--- mnuSetTargetPts.pgx ---
program mnuSetTargetPts()
  local bool LbBackup
  local num LnNewValue
  local string LsNameKeeper
  local num nKey
begin
  //header begin
  // PROGRAM mnuSetTargetPts()
  //
  // runs the menu to query user for all info needed to teach Target Frames/Points
  // with user input of Azimuth, Elevation, & Radius
  // output to X, Y, Z, RX, RY, RZ
  //
  // incoming parms:  none
  // outgoing parms:  none
  // called from:  pgm mnuTeachMenu()
  //
  //  initial release KN
  //header end
  //
  // start continuous loop, end by menu command or teach pendant command
  // on user command, jump to other subroutines for action
  //
  // init booleans for menu control in pgm displayMessage2()
  LbBackup=false
  bWorldFrameView=true
  //
  do
    //nIdxSetTargetPt=261
    call displayMessage2(nIdxSetTargetPt,nKey)
    // verify selection
    switch nKey
      // ESC key aborts, return with no save to pgm mnuTeachMenu()
      case 255
        return
      break
      // menu = Set Target Points
      // F1 to change Interaction Point number 0 or 1
      case 271
        nIPNumber=nIPNumber+1
        if nIPNumber==2
          nIPNumber=0
        endIf
      break
      // menu = Set Target Points
      // F2 to increment point number 0-19 in selected frame 0-1
      case 272
        if nIPNumber==0
          nIP1Number=nIP1Number+1
          if nIP1Number==20
            nIP1Number=0
          endIf
        else
          nIP2Number=nIP2Number+1
          if nIP2Number==20
            nIP2Number=0
          endIf
        endIf
      break
      // menu = Set Target Points, F3 to change the POINT NAME string
      // save currently selected name string to temporary variable
      // get new name string, test for >18 characters
      case 273
        gotoxy(19,3)
        put("                  ")
        gotoxy(19,3)
        if nIPNumber==0
          LsNameKeeper=sIP1TargName[nIP1Number]
          get(sIP1TargName[nIP1Number])
          if (len(sIP1TargName[nIP1Number])>18)
            popUpMsg("Name:  18 characters max...press OK")
            sIP1TargName[nIP1Number]=LsNameKeeper
          endIf
        else
          LsNameKeeper=sIP2TargName[nIP2Number]
          get(sIP2TargName[nIP2Number])
          if (len(sIP2TargName[nIP2Number])>18)
            popUpMsg("Name:  18 characters max...press OK")
            sIP2TargName[nIP2Number]=LsNameKeeper
          endIf
        endIf
        libSave()
      break
      //  menu = Set Target Points
      //  F4 ot change POINT AZIMUTH
      case 274
        // test input value for valid range
        LnNewValue=0
        gotoxy(26,4)
        get(LnNewValue)
        if LnNewValue>180 or LnNewValue<-180
          popUpMsg("ERROR:  Azimuth must be between 180 & -180 degrees...Press OK")
        else
          if nIPNumber==0
            nIP1Azimuth[nIP1Number]=LnNewValue
            //update Target Point to new AZ data
            call makePntAZELRA(nIPNumber,nIP1Number)
          else
            nIP2Azimuth[nIP2Number]=LnNewValue
            // update Target Point to new AZ data
            call makePntAZELRA(nIPNumber,nIP2Number)
          endIf
        endIf
        libSave()
      break
      // menu = Set Target Points
      // F5 to change POINT ELEVATION
      case 275
        // test input value for valid range
        LnNewValue=0
        gotoxy(26,5)
        get(LnNewValue)
        if LnNewValue>90 or LnNewValue<-90
          popUpMsg("ERROR:  Elevation must be between 90 & -90 degrees...Press OK")
        else
          if nIPNumber==0
            nIP1Elevation[nIP1Number]=LnNewValue
            // update Target Point to new EL data
            call makePntAZELRA(nIPNumber,nIP1Number)
          else
            nIP2Elevation[nIP2Number]=LnNewValue
            // update Target Point to new EL data
            call makePntAZELRA(nIPNumber,nIP2Number)
          endIf
        endIf
        libSave()
      break
      //  menu = Set Target Point (frame) Target Point
      //  F6 to change POINT RADIUS
      case 276
        //test input value for valid range
        LnNewValue=0
        gotoxy(26,6)
        get(LnNewValue)
        if LnNewValue<0
          popUpMsg("ERROR:  Negative Radius Disallowed...Press OK")
        else
          if nIPNumber==0
            nIP1Radius[nIP1Number]=LnNewValue
            // update Target Point to new RA data
            call makePntAZELRA(nIPNumber,nIP1Number)
          else
            nIP2Radius[nIP2Number]=LnNewValue
            // update Target Point to new RA data
            call makePntAZELRA(nIPNumber,nIP2Number)
          endIf
        endIf
        libSave()
      break
      // menu = Set Target Points, F7 to change displayed trsf values relative to the selected IP or World CoordSys
      // this boolean is acted upon in pgm displayMessage2()
      case 277
        if bWorldFrameView==true
          bWorldFrameView=false
        else
          bWorldFrameView=true
        endIf
      break
      //  menu = Set Target Points, F8 to save library on exit & return to pgm mnuTeachMenu()
      case 278
        libSave()
        LbBackup=true
      break
      // Any other key press
      default
        cls()
        popUpMsg("BAD SELECTION...press OK")
      break
    endSwitch
  until (false or (LbBackup==true))
  //
  // done
end

--- mnuTeachCube.pgx ---
program mnuTeachCube()
  local bool LbBackup
  local bool LbCubeAllDone
  local bool LbErrCreateCube
  local bool LbSetXYZdone
  local num LnXKeeper
  local num LnYKeeper
  local num LnZKeeper
  local point LpHere
  local string LsMoveMsg
  local num nKey
begin
  //header begin
  // PROGRAM mnuTeachCube()
  //
  // runs the menu to query user for all info needed to teach a Cubic Stay Clear Zone
  //
  // incoming parms:  none
  // outgoing parms:  none
  // called from:  pgm mnuTeachStyClr()
  //
  //  initial release KN
  //header end
  //
  // start continuous loop, end by menu command or teach pendant command
  // on user command, jump to other subroutines for action
  //
  // init booleans for menu control in pgm displayMessage1()
  LbBackup=false
  bCubeStep1=true
  bSetCylinderRZ=false
  bCylinderStep1=false
  bSetSphereRad=false
  bSphereStep1=false
  bSetCubeXYZ=false
  LbCubeAllDone=false
  // retrieve initial Cube data & store to temp variables for manipulation & display
  pOriginCube=MON:pOriginCube[nNumberCube]
  nDistXCube=MON:nDistXCube[nNumberCube]
  nDistYCube=MON:nDistYCube[nNumberCube]
  nDistZCube=MON:nDistZCube[nNumberCube]
  do
    //=========step 1==================step 1===============step 1================
    // Teach Cube, Step 1:  Tell user select and/or modify cube definitions
    do
      //nIdxTeachCube=201
      call displayMessage1(nIdxTeachCube,nKey)
      // verify selection
      switch nKey
        // ESC key aborts & returns immediately
        case 255
          return
        break
        // Teach Cube, F1 to ACCEPT definition & return to pgm mnuTeachStyClr()
        case 271
          LbCubeAllDone=true
          bSetCubeXYZ=false
          MON:nNumberCube=nNumberCube
          call MON:createCube(pOriginCube,nDistXCube,nDistYCube,nDistZCube,LbErrCreateCube)
          if LbErrCreateCube==true
            popUpMsg("Create Cube Failed...NO RECOVERY...Press OK")
            LbCubeAllDone=false
          endIf
          // saved at bottom
        break
        // menu = Teach Cube, F3 Button, change cube number via increment only
        // max = 10 as initially implemented in monitorAreaEn() library
        // max value change requires manual coordination, not automatic
        case 273
          nNumberCube=nNumberCube+1
          if nNumberCube==10
            nNumberCube=0
          endIf
          pOriginCube=MON:pOriginCube[nNumberCube]
          nDistXCube=MON:nDistXCube[nNumberCube]
          nDistYCube=MON:nDistYCube[nNumberCube]
          nDistZCube=MON:nDistZCube[nNumberCube]
        break
        // menu = Teach Cube, F4 Button, Tell user to Teach Origin Point
        case 274
          LsMoveMsg="Move SensorTool to Cube #"+toString("2.0",nNumberCube)+" Origin Point...OK to Teach"
          popUpMsg(LsMoveMsg)
          pOriginCube=here(tSensorTool,world)
        break
        //  menu = Teach Cube, F5 Button, Define DX, DY, DZ values
        case 275
          bSetCubeXYZ=true
          bCubeStep1=false
        break
        // menu = Teach Cube, F7 to reset this cube definition to {0, 0, 0}
        // this disables checking on this cube
        case 277
          MON:pOriginCube[nNumberCube].trsf={0,0,0,0,0,0}
          MON:nDistXCube[nNumberCube]=0
          MON:nDistYCube[nNumberCube]=0
          MON:nDistZCube[nNumberCube]=0
          pOriginCube.trsf={0,0,0,0,0,0}
          nDistXCube=0
          nDistYCube=0
          nDistZCube=0
          MON:nNumberCube=nNumberCube
          MON:bCreateCube[nNumberCube]=false
          MON:libSave()
          popUpMsg("CubeZone "+toString(".0",nNumberCube)+" CLEARED...Press OK")
        break
        // menu = Teach Cube, F8 Button, ABORT to Teach Stay Clear Zone Menu
        case 278
          bCubeStep1=false
          return
        break
        // Any other key press
        default
          cls()
          popUpMsg("BAD SELECTION...press OK")
        break
      endSwitch
    until (false or (bSetCubeXYZ==true) or (LbCubeAllDone==true))
    //
    //====step 2==============step 2===================step 2===============
    // menu = Teach Cube Step 2:  set the DX DY DZ values if required
    // Cube DX, DY, DZ values set here are temp to this pgm
    // only saved permanently in MON library on formal SAVE (F1) in above Step1
    if bSetCubeXYZ==true
      LbSetXYZdone=false
      do
        //nIdxSetCubeXYZ=211
        call displayMessage1(nIdxSetCubeXYZ,nKey)
        // verify selection
        switch nKey
          // ESC key aborts & returns immediately
          case 255
            return
          break
          // user accepts input from step 2 and auto backup to previous menu for acceptance
          case 271
            LbSetXYZdone=true
            bCubeStep1=true
          break
          case 274
            // user enters a new value for Cube DX
            gotoxy(25,6)
            LnXKeeper=nDistXCube
            get(nDistXCube)
            if (nDistXCube<0)
              popUpMsg("Negative values for Cube DX not allowed...Press OK")
              nDistXCube=LnXKeeper
            endIf
          break
          // user enters a new value for Cube DY
          case 275
            gotoxy(25,7)
            LnYKeeper=nDistYCube
            get(nDistYCube)
            if (nDistYCube<0)
              popUpMsg("Negative values for Cube DY not allowed...Press OK")
              nDistYCube=LnYKeeper
            endIf
          break
          // user enters a new value for Cube DZ
          case 276
            gotoxy(25,8)
            LnZKeeper=nDistZCube
            get(nDistZCube)
            if nDistZCube<0
              popUpMsg("Negative values for Cube DZ not allowed...Press OK")
              nDistZCube=LnZKeeper
            endIf
          break
          // ABORT to Teach Stay Clear Zone Menu menu and return to pgm mnuTeachStyClr()
          case 278
            bCubeStep1=false
            return
          break
          default
            popUpMsg("BAD SELECTION...Press OK")
          break
        endSwitch
      until (false or (LbSetXYZdone==true))
    endIf
    bSetCubeXYZ=false
    LbSetXYZdone=false
    //
  until (false or (LbCubeAllDone==true))
  bCubeStep1=false
  //
  // Teach Cube completed, save data on Exit
  libSave()
  MON:libSave()
  //
  //done
end

--- mnuTeachCyl.pgx ---
program mnuTeachCyl()
  local bool LbBackup
  local bool LbCylAllDone
  local bool LbErrCreateCyl
  local bool LbSetCylRZdone
  local num LnRKeeper
  local num LnZKeeper
  local point LpHere
  local string LsMoveMsg
  local num nKey
begin
  //header begin
  // PROGRAM mnuTeachCyl()
  //
  // runs the menu to query user for all info needed to teach a Cylinder Stay Clear Zone
  //
  // incoming parms:  none
  // outgoing parms:  none
  // called from:  pgm mnuTeachStyClr()
  //
  //  initial release KN
  //header end
  //
  // start continuous loop, end by menu command or teach pendant command
  // on user command, jump to other subroutines for action
  //
  // init booleans for menu control here & in displayMessage1()
  LbBackup=false
  bSetCubeXYZ=false
  bCubeStep1=false
  bSphereStep1=false
  bSetSphereRad=false
  bSetCylinderRZ=false
  bCylinderStep1=true
  LbCylAllDone=false
  // retrieve initial Cylinder data and store to temp variables for manipulation & display
  pOriginCylinder=MON:pOriginCylinder[nNumberCylinder]
  nRadiusCylinder=MON:nRadiusCylinder[nNumberCylinder]
  nDistZCylinder=MON:nDistZCylinder[nNumberCylinder]
  do
    //=========step 1==================step 1===============step 1================
    // menu = Teach Cylinder, Step 1:  Main Cylinder Info Display
    do
      //nIdxTeachCyl=221
      call displayMessage1(nIdxTeachCyl,nKey)
      // verify selection
      switch nKey
        // ESC key aborts & returns immediately
        case 255
          return
        break
        // Teach Cylinder, F1 to ACCEPT definition & return to pgm mnuTeachStyClr()
        case 271
          LbCylAllDone=true
          bSetCylinderRZ=false
          MON:nNumberCylinder=nNumberCylinder
          call MON:createCylinder(pOriginCylinder,nRadiusCylinder,nDistZCylinder,LbErrCreateCyl)
          if LbErrCreateCyl==true
            popUpMsg("Create Cylinder Failed...NO RECOVERY...Press OK")
            LbCylAllDone=false
          endIf
          // saved at bottom
        break
        // menu = Teach Cylinder, F3 Button, change cylinder number via increment only
        // max = 10 as initially implemented in monitorAreaEn() library
        // max value change requires manual coordination, not automatic
        case 273
          nNumberCylinder=nNumberCylinder+1
          if nNumberCylinder==10
            nNumberCylinder=0
          endIf
          pOriginCylinder=MON:pOriginCylinder[nNumberCylinder]
          nRadiusCylinder=MON:nRadiusCylinder[nNumberCylinder]
          nDistZCylinder=MON:nDistZCylinder[nNumberCylinder]
        break
        // menu = Teach Cylinder, F4 Button, Tell user to Teach Origin Point
        case 274
          LsMoveMsg="Move robot to Cylinder #"+toString("2.0",nNumberCylinder)+" Origin Point...OK to Teach"
          popUpMsg(LsMoveMsg)
          pOriginCylinder=here(tSensorTool,world)
        break
        //  menu = Teach Cylinder, F5 Button, goto Step2 to Define Radius & DZ values
        case 275
          bSetCylinderRZ=true
          bCylinderStep1=false
        break
        // menu = Teach Cylinder, F7 to reset this cylinder definition to {0,0,0}
        // this disables checking of this cylinder volume
        case 277
          MON:pOriginCylinder[nNumberCylinder].trsf={0,0,0,0,0,0}
          MON:nRadiusCylinder[nNumberCylinder]=0
          MON:nDistZCylinder[nNumberCylinder]=0
          pOriginCylinder.trsf={0,0,0,0,0,0}
          nRadiusCylinder=0
          nDistZCylinder=0
          MON:nNumberCylinder=nNumberCylinder
          MON:bCreateCylinder[nNumberCube]=false
          MON:libSave()
          popUpMsg("CylinderZone "+toString(".0",nNumberCylinder)+" CLEARED...Press OK")
        break
        // menu = Teach Cylinder, F8 Button, ABORT & Backup
        case 278
          bCylinderStep1=false
          return
        break
        // Any other key press
        default
          cls()
          popUpMsg("BAD SELECTION...press OK")
        break
      endSwitch
    until (false or (bSetCylinderRZ==true) or (LbCylAllDone==true))
    //
    //====step 2==============step 2===================step 2===============
    // menu = Teach Cylinder Step 2:  set the Radius & DZ values if required
    // Cylinder DZ & Radius values here are temp to this pgm
    // only saved permanently in MON library on formal SAVE (F1) in above Step1
    if bSetCylinderRZ==true
      LbSetCylRZdone=false
      do
        //nIdxSetCylRZ=231
        call displayMessage1(nIdxSetCylRZ,nKey)
        // verify selection
        switch nKey
          // ESC key aborts & returns immediately
          case 255
            return
          break
          // user accepts Cylinder Radius & Z-Distance input from step 2 and...
          // auto backup to previous menu for acceptance
          case 271
            LbSetCylRZdone=true
            bCylinderStep1=true
          break
          case 274
            // user enters a new value for Cylinder Radius
            gotoxy(30,6)
            LnRKeeper=nRadiusCylinder
            get(nRadiusCylinder)
            if (nRadiusCylinder<0)
              popUpMsg("Negative values disallowed...Press OK")
              nRadiusCylinder=LnRKeeper
            endIf
          break
          // user enters a new value for Cylinder DZ
          case 275
            gotoxy(25,7)
            LnZKeeper=nDistZCylinder
            get(nDistZCylinder)
            if nDistZCylinder<0
              popUpMsg("Negative values disallowed...Press OK")
              nDistZCylinder=LnZKeeper
            endIf
          break
          // menu Teach Cylinder, F7 to clear this cylinder definition
          // this disables checking of this cylinder volume
          case 277
            MON:pOriginCylinder[nNumberCylinder].trsf={0,0,0,0,0,0}
            MON:nRadiusCylinder[nNumberCylinder]=0
            MON:nDistZCylinder[nNumberCylinder]=0
            pOriginCylinder.trsf={0,0,0,0,0,0}
            nRadiusCylinder=0
            nDistZCylinder=0
            MON:nNumberCylinder=nNumberCylinder
            MON:libSave()
          break
          // ABORT & backup to previous menu
          case 278
            bCylinderStep1=false
            return
          break
          // any other key press
          default
            cls()
            popUpMsg("BAD SELECTION...Press OK")
          break
        endSwitch
      until (false or (LbSetCylRZdone==true))
    endIf
    bSetCylinderRZ=false
    LbSetCylRZdone=false
    //
  until (false or (LbCylAllDone==true))
  bCylinderStep1=false
  //
  // Teach Cylinder completed, save data on exit
  //
  libSave()
  MON:libSave()
  //
  // done
end

--- mnuTeachFrame.pgx ---
program mnuTeachFrame()
  local bool LbTeachFrm1of5
  local bool LbTeachFrm2of5
  local bool LbTeachFrm3of5
  local bool LbTeachFrm4of5
  local bool LbTeachFrm5of5
  local point LpFrameOrigin
  local point LpFrameXAxis
  local point LpFrameYAxis
  local num nKey
begin
  //header begin
  // PROGRAM mnuTeachFrame()
  //
  // runs the Wizard to assist user:  Teach the Target Frame of the two targets
  //
  // incoming parms:  none
  // outgoing parms:  none
  // called from:  pgm mnuTeachIP()
  //
  //  initial release KN
  //  Release 2 KN
  //    this pgm now called from pgm mnuTeachIP()
  //
  //header end
  //
  // start continuous loop, go through each of 5 wizard steps
  //
  // init step-by-step continuance booleans
  LbTeachFrm1of5=false
  LbTeachFrm2of5=false
  LbTeachFrm3of5=false
  LbTeachFrm4of5=false
  LbTeachFrm5of5=false
  //
  // menu = Teach Interaction Point Frame, Step 1 of 5 Steps:  select the frame to be taught
  do
    // nIdxFrm1of5=131
    call displayMessage(nIdxFrm1of5,nKey)
    // verify selection
    switch nKey
      // ESC aborts & returns immediately
      case 255
        return
      break
      // menu = Teach Interaction Point Frame 1of5, F1 to continue to Step 2 of 4
      case 271
        LbTeachFrm1of5=true
      break
      // menu = Teach Interaction Point Frame 1of5, F3 Button, user changes Target Number
      case 273
        if nIPNumber==1
          nIPNumber=-1
        else
          nIPNumber=nIPNumber+1
        endIf
      break
      // menu = Teach Interaction Point Frame 1of5, F8 Button, ABORT & backup to Teach Menu
      case 278
        return
      break
      // Any other key press
      default
        popUpMsg("BAD SELECTION...press OK")
      break
    endSwitch
  until (false or (LbTeachFrm1of5==true))
  //
  // menu = Teach Interaction Point Frame, Step 2 of 5 Steps:  verify Ref Pointer tool is attached
  do
    // nIdxFrm2of5=141
    call displayMessage(nIdxFrm2of5,nKey)
    // verify selection
    switch nKey
      // ESC key aborts & returns immediately
      case 255
        return
      break
      // menu = Teach Interaction Point Frame 2of5, F1 to continue to Step 3 of 5
      case 271
        LbTeachFrm2of5=true
      break
      // menu = Teach Interaction Point Frame 2of5, F8 Button, ABORT & backup to Teach Menu
      case 278
        return
      break
      // Any other key press
      default
        popUpMsg("BAD SELECTION...press OK")
      break
    endSwitch
  until (false or (LbTeachFrm2of5==true))
  //
  // menu = Teach Interaction Point Frame, Step 3 of 5 Steps:  move to Frame Origin
  do
    // nIdxFrm3of5=151
    call displayMessage(nIdxFrm3of5,nKey)
    // verify selection
    switch nKey
      // ESC key aborts & returns immediately
      case 255
        return
      break
      // menu = Teach Interaction Point Frame 3of5, F1 Button, teach frame origin point
      case 271
        LpFrameOrigin=here(tRefPointer,world)
        LbTeachFrm3of5=true
      break
      // menu = Teach Interaction Point Frame 3of5, F8 Button, ABORT & backup to Teach Menu
      case 278
        return
      break
      // Any other key press
      default
        popUpMsg("BAD SELECTION...press OK")
      break
    endSwitch
  until (false or (LbTeachFrm3of5==true))
  //
  // menu = Teach Interaction Point Frame, Step 4 of 5 Steps:  teach Frame X-Axis location
  do
    // nIdxFrm4of5=161
    call displayMessage(nIdxFrm4of5,nKey)
    // verify selection
    switch nKey
      // ESC key aborts & returns immediately
      case 255
        return
      break
      // menu = Teach Interaction Point Frame 4of5, F1 Button, teach Frame X-Axis point
      case 271
        LpFrameXAxis=here(tRefPointer,world)
        LbTeachFrm4of5=true
      break
      // menu = Teach Interaction Point Frame 4of5, F8 Button, ABORT & backup to Teach Menu
      case 278
        return
      break
      // Any other key press
      default
        popUpMsg("BAD SELECTION...press OK")
      break
    endSwitch
  until (false or (LbTeachFrm4of5==true))
  //
  // menu = Teach Interaction Point Frame, Step 5 of 5 Steps:  Teach Frame y-Axis direction point
  do
    // nIdxFrm5of5=171
    call displayMessage(nIdxFrm5of5,nKey)
    // verify selection
    switch nKey
      // ESC key aborts & returns immediately
      case 255
        return
      break
      // menu = Teach Interaction Point Frame 5of5, F1 Button, User Accepts Frame definition
      case 271
        LpFrameYAxis=here(tRefPointer,world)
        if nIPNumber==-1
          setFrame(LpFrameOrigin,LpFrameXAxis,LpFrameYAxis,fIPoriginal)
        elseIf nIPNumber==0
          setFrame(LpFrameOrigin,LpFrameXAxis,LpFrameYAxis,fIP1)
        elseIf nIPNumber==1
          setFrame(LpFrameOrigin,LpFrameXAxis,LpFrameYAxis,fIP2)
        endIf
        LbTeachFrm5of5=true
      break
      // menu = Teach Interaction Point Frame 5of5, F8 Button, ABORT & backup to Teach Menu
      case 278
        return
      break
      // Any other key press
      default
        popUpMsg("BAD SELECTION...press OK")
      break
    endSwitch
  until (false or (LbTeachFrm5of5==true))
  //
  // teach Interaction Point Frame completed, save data on exit
  libSave()
  //
  // done
end

--- mnuTeachIP.pgx ---
public program mnuTeachIP()
  local bool LbBackup
  local num nKey
begin
  //header begin
  // PROGRAM mnuTeachP()
  //
  // runs the menu to Teach the Interaction Point by two methods:
  //    (1) Direct Entry of Interaction Point {X, Y, Z, RX, RY, RZ} values
  //    (2) Use a Wizard to walk through the steps to physically teach the IP with a reference pointer tool
  //
  // incoming parms:  none
  // outgoing parms:  none
  // called from:  pgm mnuTeachMenu()
  //
  //  this program is part of SLAC Release 2:  KN
  //
  //header end
  //
  // start continuous loop, end by menu command or teach pendant command
  // on user command, jump to other subroutines for action
  //
  LbBackup=false
  do
    // nIdxTeachIP = 331
    call displayMessage6(nIdxTeachIP,nKey)
    // verify selection
    switch nKey
      // ESC key aborts & returns immediately
      case 255
        return
      break
      // menu = Teach TCP:  F1 Button, Toggle selection of Interaction Point Number
      case 271
        if nIPNumber==1
          nIPNumber=-1
        else
          nIPNumber=nIPNumber+1
        endIf
      break
      // menu = Teach TCP:  F2 Button, Direct Entry of Interaction Point {X, Y, Z, RX, RY, RZ} values
      case 272
        call mnuEnterIPVals()
      break
      // menu = Teach TCP:  F3 Button, run Wizard to Teach Interaction Point with reference pointer
      case 273
        call mnuTeachFrame()
      break
      //  menu = Teach TCP:  F8 Button, backup to Teach Menu
      case 278
        LbBackup=true
      break
      // ALL OTHER CHOICES
      default
        popUpMsg("mnuTeachIP:  BAD SELECTION...Press OK")
      break
    endSwitch
  until (false or (LbBackup==true))
  // done
  if nIPNumber==-1
    nIPNumber=0
  endIf
end

--- mnuTeachMenu.pgx ---
program mnuTeachMenu()
  local bool LbBackup
  local num nKey
begin
  //header begin
  // PROGRAM mnuTeachMenu()
  //
  // runs the menu to select various TEACH functions
  //
  // incoming parms:  none
  // outgoing parms:  none
  // called from:  pgm main()
  //
  //  initial release KN
  //  Release 2  KN
  //    changed F2 to call pgm mnuTeachIP() for different Teach IP methods
  //
  //header end
  //
  // start continuous loop, end by menu command or teach pendant command
  // on user command, jump to other subroutines for action
  //
  LbBackup=false
  do
    // nIdxTeachMenu = 11
    call display(nIdxTeachMenu,nKey)
    // verify selection
    switch nKey
      // ESC key aborts & returns immediately
      case 255
        LbBackup=true
      break
      // menu = Teach Menu:  F1 Teach & Edit Target Points
      case 271
        call mnuSetTargetPts()
      break
      // menu = Teach Menu:  F2 Button, go to menu for different Teach IP functions
      case 272
        call mnuTeachIP()
      break
      // menu = Teach Menu:  F3 Button, Teach PARK Location
      case 273
        call mnuTeachPark()
      break
      // menu = Teach Menu:  F4 Button, Teach PARK TOP Location
      case 274
        call mnuTeachParkTop()
      break
      // menu = Teach Menu:  F5 Button, Teach TCP
      case 275
        call mnuTeachTCP()
      break
      // menu = Teach Menu:  F6 Button, Teach Stay Clear zones
      case 276
        call mnuTeachStayClr()
      break
      // menu = Teach Menu:  F8 Button, backup to Main Menu
      case 278
        LbBackup=true
      break
      // any other key press
      default
        cls()
        popUpMsg("BAD SELECTION...Press OK")
      break
    endSwitch
  until (false or (LbBackup==true))
  // done
end

--- mnuTeachPark.pgx ---
program mnuTeachPark()
  local bool LbBackup
  local num nKey
begin
  //header begin
  // PROGRAM mnuTeachPark()
  //
  // runs the Wizard to assist user:  Teach a single robot PARK position
  // position taught = jPark
  //
  // incoming parms:  none
  // outgoing parms:  none
  // called from:  pgm mnuTeachMenu()
  //
  //  initial release KN
  //header end
  //
  // start continuous loop, go through each of 5 wizard steps
  //
  // init step-by-step continuance booleans
  LbBackup=false
  //
  do
    // nIdxTeachPARK=51
    call displayMessage(nIdxTeachPARK,nKey)
    // verify selection
    switch nKey
      // ESC key aborts & returns immediately
      case 255
        return
      break
      // menu = Teach Park, F1 to continue to Step 2 of 4
      case 271
        jPark=herej()
        LbBackup=true
      break
      // menu = Teach Park, F8 Button, abort to Teach Menu
      case 278
        return
      break
      // Any other key press
      default
        popUpMsg("BAD SELECTION...press OK")
      break
    endSwitch
  until (false or (LbBackup==true))
  //
  // teach Park Position completed, save data on exit
  libSave()
  //
  // done
end

--- mnuTeachParkTop.pgx ---
program mnuTeachParkTop()
  local bool LbBackup
  local num nKey
begin
  //header begin
  // PROGRAM mnuTeachPark()
  //
  // runs the Wizard to assist user:  Teach a single robot PARK position
  // position taught = jPark
  //
  // incoming parms:  none
  // outgoing parms:  none
  // called from:  pgm mnuTeachMenu()
  //
  //  initial release KN
  //header end
  //
  // start continuous loop, go through each of 5 wizard steps
  //
  // init step-by-step continuance booleans
  LbBackup=false
  //
  do
    // nIdxTeachPARKTOP=371
    call displayMessage(nIdxTeachPARKT,nKey)
    // verify selection
    switch nKey
      // ESC key aborts & returns immediately
      case 255
        return
      break
      // menu = Teach Park, F1 to continue to Step 2 of 4
      case 271
        jParkTop=herej()
        LbBackup=true
      break
      // menu = Teach Park, F8 Button, abort to Teach Menu
      case 278
        return
      break
      // Any other key press
      default
        popUpMsg("BAD SELECTION...press OK")
      break
    endSwitch
  until (false or (LbBackup==true))
  //
  // teach Park Position completed, save data on exit
  libSave()
  //
  // done
end

--- mnuTeachSphere.pgx ---
program mnuTeachSphere()
  local bool LbBackup
  local bool LbErrCreateSph
  local bool LbSetSphRdone
  local bool LbSphAllDone
  local num LnRKeeper
  local point LpHere
  local string LsMoveMsg
  local num nKey
begin
  //header begin
  // PROGRAM mnuTeachSphere()
  //
  // runs the menu to query user for all info needed to teach a Sphere Stay Clear Zone
  //
  // incoming parms:  none
  // outgoing parms:  none
  // called from:  pgm mnuTeachStyClr()
  //
  //  initial release KN
  //header end
  //
  // start continuous loop, end by menu command or teach pendant command
  // on user command, jump to other subroutines for action
  //
  // init booleans for menu control here & in pgm displayMessage1()
  LbBackup=false
  bSetCubeXYZ=false
  bCubeStep1=false
  bSetCylinderRZ=false
  bCylinderStep1=false
  bSetSphereRad=false
  bSphereStep1=true
  LbSphAllDone=false
  // retrieve initial Cyl data & store to temp variables for manipulation & display
  pOriginSphere=MON:pOriginSphere[nNumberSphere]
  nRadiusSphere=MON:nRadiusSphere[nNumberSphere]
  do
    //=========step 1==================step 1===============step 1================
    // menu = Teach Sphere, Step 1:  Main Sphere Info Display
    do
      //nIdxTeachSph=241
      call displayMessage1(nIdxTeachSph,nKey)
      // verify selection
      switch nKey
        // ESC key aborts & returns immediately
        case 255
          return
        break
        // menu = Teach Sphere, F1 to ACCEPT definition & return to pgm mnuTeachStyClr()
        case 271
          LbSphAllDone=true
          MON:nNumberSphere=nNumberSphere
          call MON:createSphere(pOriginSphere,nRadiusSphere,LbErrCreateSph)
          if LbErrCreateSph==true
            popUpMsg("Create Sphere Failed...Press OK")
            LbSphAllDone=false
          endIf
          // saved at bottom
        break
        // menu = Teach Sphere, F3 Button, change sphere number via increment only
        // max = 10 as initially implemented in monitorAreaEn() library
        // max value change requires manual coordination, not automatic
        case 273
          nNumberSphere=nNumberSphere+1
          if nNumberSphere==10
            nNumberSphere=0
          endIf
          pOriginSphere=MON:pOriginSphere[nNumberSphere]
          nRadiusSphere=MON:nRadiusSphere[nNumberSphere]
        break
        // menu = Teach Sphere, F4 Button, Tell user to Teach Origin Point
        case 274
          LsMoveMsg="Move robot to Sphere #"+toString("2.0",nNumberSphere)+" Origin Point...OK to Teach"
          popUpMsg(LsMoveMsg)
          pOriginSphere=here(tSensorTool,world)
        break
        //  menu = Teach Sphere, F5 Button, goto next step to Define Radius
        case 275
          bSetSphereRad=true
          bSphereStep1=false
        break
        // menu = Teach Sphere, F7 clears the current sphere definition
        // this disables the checking of the sphere
        case 277
          MON:pOriginSphere[nNumberSphere].trsf={0,0,0,0,0,0}
          MON:nRadiusSphere[nNumberSphere]=0
          pOriginSphere.trsf={0,0,0,0,0,0}
          nRadiusSphere=0
          MON:nNumberSphere=nNumberSphere
          MON:bCreateSphere[nNumberSphere]=false
          MON:libSave()
          popUpMsg("SphereZone "+toString(".0",nNumberSphere)+" CLEARED...Press OK")
        break
        // menu = Teach Sphere, F8 Button, ABORT & Backup
        case 278
          bSphereStep1=false
          return
        break
        // Any other key press
        default
          cls()
          popUpMsg("BAD SELECTION...press OK")
        break
      endSwitch
    until (false or (bSetSphereRad==true) or (LbSphAllDone==true))
    //
    //====step 2==============step 2===================step 2===============
    // menu = Teach Sphere Step 2:  set the Radius
    // Sphere DZ & Radius values here are temp to this pgm
    // only permanently saved to MON library on formal SAVE (F1) in above Step1
    if bSetSphereRad==true
      LbSetSphRdone=false
      do
        //nIdxSetSphRad=251
        call displayMessage1(nIdxSetSphRad,nKey)
        // verify selection
        switch nKey
          // ESC key aborts & returns immediately
          case 255
            return
          break
          // user accepts input from step 2 and auto backup to previous menu for accept and save
          case 271
            LbSetSphRdone=true
            bSphereStep1=true
          break
          case 274
            // user enters a new value for Sphere Radius
            gotoxy(30,6)
            LnRKeeper=nRadiusSphere
            get(nRadiusSphere)
            if (nRadiusSphere<0)
              popUpMsg("Negative values disallowed...Press OK")
              nRadiusSphere=LnRKeeper
            endIf
          break
          // ABORT & backup to previous pgm mnuSetStyClr()
          case 278
            bSphereStep1=false
            return
          break
          // any other key press
          default
            cls()
            popUpMsg("BAD SELECTION...Press OK")
          break
        endSwitch
      until (false or (LbSetSphRdone==true))
    endIf
    bSetSphereRad=false
    LbSetSphRdone=false
    //
  until (false or (LbSphAllDone==true))
  bSphereStep1=false
  //
  // Teach Sphere completed, save data on exit
  //
  libSave()
  MON:libSave()
  //
  // done
end

--- mnuTeachStayClr.pgx ---
program mnuTeachStayClr()
  local bool LbBackup
  local num nKey
begin
  //header begin
  // PROGRAM mnuTeachStayClr()
  //
  // runs the menu to select which type of Stay Clear Area to Teach
  // Cube, Cylinder, or Sphere
  //
  // incoming parms:  none
  // outgoing parms:  none
  // called from:  pgm mnuTeachMenu()
  //
  //  initial release KN
  //header end
  //
  // start continuous loop, end by menu command or teach pendant command
  // on user command, jump to other subroutines for action
  //
  LbBackup=false
  do
    // nIdxStyClr=61
    call display(nIdxStyClr,nKey)
    // verify selection
    switch nKey
      // ESC key aborts & returns immediately
      case 255
        return
      break
      // menu = Teach Stay Clear Area Menu:  F1 Button, Select Cubic Stay Clear Zone
      case 271
        call mnuTeachCube()
      break
      // menu = Teach Stay Clear Area Menu:  F2 Button, Select Cylinder Stay Clear Zone
      case 272
        call mnuTeachCyl()
      break
      // menu = Teach Stay Clear Area Menu:  F3 Button, Select Spherical Stay Clear Zone
      case 273
        call mnuTeachSphere()
      break
      //  menu = Teach Stay Clear Area Menu:  F8 Button, ABORT to Teach Menu
      case 278
        LbBackup=true
      break
      // any other key press
      default
        cls()
        popUpMsg("BAD SELECTION...Press OK")
      break
    endSwitch
  until (false or (LbBackup==true))
  // done
end

--- mnuTeachTCP.pgx ---
public program mnuTeachTCP()
  local bool LbBackup
  local num nKey
begin
  //header begin
  // PROGRAM mnuTeachTCP()
  //
  // runs the menu to select Teach TCP by pointer tool
  //
  // incoming parms:  none
  // outgoing parms:  none
  // called from:  pgm mnuTeachMenu()
  //
  //  initial release KN
  //  Release 2:  KN
  //    added Direct Entry of TCP values {X, Y, Z, RX, RY, RZ} via MCP
  //
  //header end
  //
  // start continuous loop, end by menu command or teach pendant command
  // on user command, jump to other subroutines for action
  //
  LbBackup=false
  do
    // nIdxTeachTCP = 21
    call display(nIdxTeachTCP,nKey)
    // verify selection
    switch nKey
      // ESC key aborts & returns immediately
      case 255
        return
      break
      // menu = Teach TCP:  F1 Button, Teach TCP with pointer tool
      case 271
        call mnuTeachTCPptr()
      break
      // menu = Teach TCP:  F2 Button, Teach TCP with 4-point method
      case 272
        call mnuTeachTCP4pnt()
      break
      // menu = Teach TCP:  F3 Button, Direct Entry of TCP values {X, Y, Z, RX, RY, RZ}
      case 273
        call mnuEnterTCPVals()
      break
      //  menu = Teach TCP:  F8 Button, backup to Teach Menu
      case 278
        LbBackup=true
      break
      // ALL OTHER CHOICES
      default
        popUpMsg("BAD SELECTION...Press OK")
      break
    endSwitch
  until (false or (LbBackup==true))
  // done
end

--- mnuTeachTCP4pnt.pgx ---
program mnuTeachTCP4pnt()
begin
  //header begin
  // PROGRAM mnuTeachTCP4pnt()
  //
  // runs the menu to Teach the EOAT TCP by use of 4-point teach method
  // call Staubli-supplied library CalcTool4pEn(), used here with
  // minor modifications
  //
  // incoming parms:  none
  // outgoing parms:  none
  // called from:  pgm mnuTeachTCP()
  //
  //  initial release KN
  //header end
  //
  // library TCP4:calcTool4pEN is AUTOLOADED
  call TCP4:aMainTcp(100)
  // take the trsf calculated by the 4-point routine and use it for the SLAC sensor tool
  tSensorTool.trsf=trUserTool
  //
  // teach new tool def with 4-pnt method completed, save data on exit
  libSave()
  // done
end

--- mnuTeachTCPptr.pgx ---
program mnuTeachTCPptr()
  local bool LbTeachTCP1of4
  local bool LbTeachTCP2of4
  local bool LbTeachTCP3of4
  local bool LbTeachTCP4of4
  local point LpHere
  local num nKey
begin
  //header begin
  // PROGRAM mnuTeachTCPptr()
  //
  // runs the menu to Teach the EOAT TCP by use of "ptr" pointer tool
  // provides a "Wizard" to assist the user through manual steps required
  //
  // incoming parms:  none
  // outgoing parms:  none
  // called from:  pgm mnuTeachTCP()
  //
  //  initial release KN
  //header end
  //
  // start continuous loop, end by menu command or teach pendant command
  // on user command, jump to other subroutines for action
  //
  // init local step-by-step continuance booleans
  //
  LbTeachTCP1of4=false
  LbTeachTCP2of4=false
  LbTeachTCP3of4=false
  LbTeachTCP4of4=false
  //
  //=========================================================================================
  // Teach TCP with Pointer, Step 1 of 4 Steps:  verify pointer tool & Cell Reference Pointer
  do
    // nIdxTCP1of4=81
    call displayMessage(nIdxTCP1of4,nKey)
    // verify selection
    switch nKey
      // ESC key aborts & returns immediately
      case 255
        return
      break
      // menu = Teach TCP with pointer 1of4, F1 to continue to Step 2 of 4
      case 271
        LbTeachTCP1of4=true
      break
      // menu = Teach TCP with pointer 1of4, F8 Button, ABORT to Teach TCP Menu
      case 278
        return
      break
      // Any other key press
      default
        popUpMsg("BAD SELECTION...press OK")
      break
    endSwitch
  until (false or (LbTeachTCP1of4==true))
  //
  //=====================================================================================
  // Teach TCP with Pointer, Step 2 of 4 Steps:  move to Cell Reference with Pointer Tool
  do
    LbTeachTCP1of4=false
    // nIdxTCP2of4=91
    call displayMessage(nIdxTCP2of4,nKey)
    // verify selection
    switch nKey
      // ESC key aborts & returns immediately
      case 255
        return
      break
      // menu = Teach TCP with pointer 2of4, F1 Button, Continue to Step 3 of 4
      // define the Cell Reference location pCellReference with pointer tool
      case 271
        pCellReference=here(tRefPointer,world)
        LpHere=here(flange,world)
        LbTeachTCP2of4=true
      break
      // menu = Teach TCP with pointer 2of4, F8 Button, ABORT to Teach TCP Menu
      case 278
        return
      break
      // Any other key press
      default
        popUpMsg("BAD SELECTION...press OK")
      break
    endSwitch
  until (false or (LbTeachTCP2of4==true))
  //
  //===================================================================================================
  // menu = Teach TCP with Pointer, Step 3 of 4 Steps:  Remove Pointer, Attach Sensor, Move to Cell Ref
  do
    LbTeachTCP2of4=false
    // nIdxTCP3of4=101
    call displayMessage(nIdxTCP3of4,nKey)
    // verify selection
    switch nKey
      // ESC key aborts & returns immediately
      case 255
        return
      break
      // menu = Teach TCP with pointer 3of4, F1 Button, calculate the new tool transform
      case 271
        tSensorTool.trsf=!LpHere.trsf*pCellReference.trsf
        LbTeachTCP3of4=true
      break
      // menu = Teach TCP with pointer 3of4, F8 Button, ABORT to Teach TCP Menu
      case 278
        return
      break
      // Any other key press
      default
        popUpMsg("BAD SELECTION...press OK")
      break
    endSwitch
  until (false or (LbTeachTCP3of4==true))
  //
  //=====================================================================================
  // menu = Teach TCP with Pointer, Step 4 of 4 Steps:  Verify new Sensor tool definition
  do
    LbTeachTCP3of4=false
    // nIdxTCP4of4=111
    call displayMessage(nIdxTCP4of4,nKey)
    // verify selection
    switch nKey
      // ESC key aborts & returns immediately
      case 255
        return
      break
      // menu = Teach TCP with pointer 4of4, F1 Button, User Accepts tool definition
      case 271
        LbTeachTCP4of4=true
      break
      // menu = Teach TCP with pointer 4of4, F8 Button, ABORT to Teach TCP Menu
      case 278
        return
      break
      // Any other key press
      default
        popUpMsg("BAD SELECTION...press OK")
      break
    endSwitch
  until (false or (LbTeachTCP4of4==true))
  //
  LbTeachTCP4of4=false
  // teach new tool def completed, save data on normal exit of this program
  libSave()
  // done
end

--- mnuTestSimESTOP.pgx ---
program mnuTestSimESTOP()
  local bool LbDone
  local num nKey
begin
  //header begin
  // PROGRAM mnuTestSimESTOP()
  //
  // runs the menu to test for bSimulateESTOP is on, get user to continue or disable
  //
  // incoming parms:  none
  // outgoing parms:  none
  // called from:  pgm main()
  //
  //  This program is released as part of SLAC RX130L robot control code Revision 3.
  //  This is part of Blue Technik proposal K01c
  //header end
  //
  // start continuous loop, end by menu command or teach pendant command
  // on user command, jump to other subroutines for action
  //
  // init booleans for menu control in pgm displayMessage2()
  LbDone=false
  //
  do
    //
    call displayMessage9(361,nKey)
    // verify selection
    switch nKey
      // F1 to continue with bSimulateESTOP=true as initialized
      case 271
        LbDone=true
      break
      //  F8 to disable Simulated ESTOP function and continue with program
      case 278
        bSimulateESTOP=false
        LbDone=true
      break
      // Any other key press
      default
        cls()
        //
      break
    endSwitch
  until (false or (LbDone==true))
  //
  // done
end

--- mnuUtility.pgx ---
program mnuUtility()
  local bool LbBackup
  local num nKey
begin
  //header begin
  // PROGRAM menuUtility()
  //
  // runs the menu to select various functions
  //
  // incoming parms:  none
  // outgoing parms:  none
  // called from:  pgm main()
  //
  //  initial release KN
  //header end
  //
  // start continuous loop, end by menu command or teach pendant command
  // on user command, jump to other subroutines for action
  //
  LbBackup=false
  do
    // display different Utility Menus depending upon status of Zone Monitoring enable/disable
    if bStopAllMonitor==true
      // nIdxUtilityMenu = 71, shows ENABLE monitoring
      call display(nIdxUtilityMenu,nKey)
    else
      //nIdxUtilMenu2=301, shows DISABLE monitoring
      call display(nIdxUtilMenu2,nKey)
    endIf
    // verify selection
    switch nKey
      // ESC key aborts & returns immediately
      case 255
        return
      break
      // menu = Utility Menu:  F1 Button = Initialize Robot
      case 271
        call initializeRobot()
      break
      // menu = Utility Menu:  F2 Button = Verify arm is at Park, option to user to move arm even if not at park
      case 272
        call checkAtPark()
      break
      // menu = Utility Menu:  F3 Button to change enable/disable status of Stay Clear Zone checking
      case 273
        if bStopAllMonitor==false
          bStopAllMonitor=true
        else
          bStopAllMonitor=false
        endIf
      break
      // menu = Utility Menu, F4 to allow user to set global speed
      case 274
        call mnuGlobalSpeed()
      break
      // menu = Utility Menu:  F5 Button, ENABLE Remote Control of Robot Functions from Host Computer
      // boolean bRemControlON used inside of tskRemControl()
      case 275
        bRemControlON=true
        do
          delay(1)
        until bRemControlON==false
        //
      break
      // menu = Utility Menu:  F6 Button, Display to User Page TCP locations relative to
      // /selected Interaction Point frame
      case 276
        call mnuGetTCP()
      break
      // menu = Utility Menu:  F8 Button, backup to Main Menu
      case 278
        LbBackup=true
      break
      // any other key press
      default
        cls()
        popUpMsg("BAD SELECTION...Press OK")
      break
    endSwitch
  until (false or (LbBackup==true))
  // done
end

--- movTargetPoint.pgx ---
public program movTargetPoint()
  local num LnDistToPark
  local num LnDistToTP
  local num LnDistance
  local num LnKey
  local point LpHere
  local point LpPark
  local point LpTargetPoint
begin
  //header begin
  // PROGRAM movTargPoint()
  //
  // checks for necessary conditions to be met before move to
  // currently selected Target Point at currently selected Interaction Point
  //
  // incoming parms:  none
  // outgoing parms:  none
  // called from:  pgm mnuMoveTargPnt()
  //
  //  initial release KN
  //header end
  //
  //
  // stop all current moves and clear motion stack
  stopMove()
  resetMotion()
  // test for ESTOP, Manual Mode, Arm Power, & Arm Cal
  call initializeRobot()
  //
  cls()
  title(" MOVE TO TARGET POINT ")
  //
  // test if "near to" currently selected Target Point in case user desires return from adjustment loc to Target Point
  LpHere=here(tSensorTool,world)
  if nIPNumber==0
    LpTargetPoint=pIP1Point[nIP1Number]
  else
    LpTargetPoint=pIP2Point[nIP2Number]
  endIf
  LnDistToTP=abs(distance(LpHere,LpTargetPoint))
  logMsg("dist to TP="+toString(".2",LnDistToTP))
  //
  // Test if arm not close enough to Target Point, then test for distance to jPark
  // check if arm is at pre-defined jPark location, deny motion & advise user & return if not at jPark
  // get current position, compare with destination
  LpHere=here(tSensorTool,world)
  LpPark=jointToPoint(tSensorTool,world,jPark)
  LnDistToPark=abs(distance(LpHere,LpPark))
  logMsg("Dist to Park="+toString(".2",LnDistToPark))
  // if arm is close enough to TP to safely move back to TP, or is close enough to jPark to safely move to TP, then move
  // else deny motion
  if ((LnDistToTP<=nAdjPntMoveTol) or (LnDistToPark<=nParkTolerance))
    // if arm is close enough to Target Point or to jPark, then go ahead and move to Target Point
    //
    gotoxy(0,4)
    putln("WAITING:  Push MOVE/HOLD")
    putln("          to move to Target Point")
    // put "HALT" in F8 position
    gotoxy(36,13)
    put("HALT")
    //
    bEnableMonitor=true
    if nIPNumber==0
      movej(pIP1Point[nIP1Number],tSensorTool,mGlobalSpeed)
      LpTargetPoint=pIP1Point[nIP1Number]
    else
      movej(pIP2Point[nIP2Number],tSensorTool,mGlobalSpeed)
      LpTargetPoint=pIP2Point[nIP2Number]
    endIf
    // watch for Stay Clear Zone entry, process if required
    // watch for bStopMotion initiated from tskHaltMoveMon()
    bWatchForHalt=true
    do
      // get current position, compare with destination
      LpHere=here(tSensorTool,world)
      LnDistance=abs(distance(LpHere,LpTargetPoint))
      delay(0)
      // exits do-until loop if TCP within tolerance of destination point or if F8=HALT key is pressed during motion
    until (LnDistance<=nZoneWatchTol) or (bInsideCube==true) or (bInsideCylinder==true) or (bInsideSphere==true) or (bStopMotion==true)
    //
    // if within tolerance zone, continue on until end of move at Target Point
    if (bInsideCube==false) and (bInsideCylinder==false) and (bInsideSphere==false) and (LnDistance<=nZoneWatchTol) and (bStopMotion==false)
      waitEndMove()
      popUpMsg("NOW at Target Point...Press OK")
      logMsg("movTargetPoint():  target point move complete")
      //...else there is a stopping condition of TCP inside a Stay Clear Zone or F8=HALT button is pressed during motion
    else
      stopMove()
      resetMotion()
      bStopAllMonitor=true
      popUpMsg("MOTION CANCELLED:  Zone Entered or HALT requested; Monitoring is Disabled; Manual Recovery REQUIRED...Press OK")
      logMsg("movTargetPoint():  zone entered or HALT requested during move")
      //
      // put in motion halt recovery steps here
      //
    endIf
  else
    popUpMsg("MOTION CANCELLED:  Arm is not close enough to Target Point or NOT PARKED...Press OK")
    logMsg("movTargetPoint():  motion cancelled due, TCP out of target point tolerance or NOT PARKED")
  endIf
  bEnableMonitor=false
  bWatchForHalt=false
  bStopMotion=false
  //
  //done
  //
end

--- movToPark.pgx ---
program movToPark()
  local num LnDistance
  local point LpHere
  local point LpPark
begin
  //
  //header begin
  //
  //header end
  //
  stopMove()
  resetMotion()
  // check robot condition:  ESTOP clear, MANUAL MODE, CALIBRATED=true, ARM POWER=ON
  call initializeRobot()
  userPage()
  cls()
  title(" MOVE TO PARK ")
  gotoxy(0,4)
  putln("WAITING:  Press MOVE/HOLD button")
  putln("          to move to Park...")
  // put "HALT" in F8 position
  gotoxy(36,13)
  put("HALT")
  //
  //
  bEnableMonitor=true
  LpPark=jointToPoint(tSensorTool,world,jPark)
  movel(LpPark,tSensorTool,mGlobalSpeed)
  //
  // watch for Stay Clear Zone entry, process if required
  // watch for bStopMotion initiated from tskHaltMoveMon()
  bWatchForHalt=true
  do
    // get current position, compare with destination
    LpHere=here(tSensorTool,world)
    LpPark=jointToPoint(tSensorTool,world,jPark)
    LnDistance=abs(distance(LpHere,LpPark))
    delay(0)
  until (LnDistance<=nZoneWatchTol) or (bInsideCube==true) or (bInsideCylinder==true) or (bInsideSphere==true) or (bStopMotion==true)
  //
  if (bInsideCube==false) and (bInsideCylinder==false) and (bInsideSphere==false) and (bStopMotion==false)
    waitEndMove()
    popUpMsg("NOW at PARK...Press OK")
  else
    stopMove()
    resetMotion()
    bStopAllMonitor=true
    popUpMsg("MOTION CANCELLED:  Zone Entered or HALT requested; Monitoring Disabled; Manual Recovery REQUIRED...Press OK")
    //
    // put in motion halt recovery steps here
    //
  endIf
  bEnableMonitor=false
  bWatchForHalt=false
  bStopMotion=false
  //
  //
  //done
  //
end

--- movToParkTop.pgx ---
program movToParkTop()
  local num LnDistance
  local point LpHere
  local point LpPark
begin
  //
  //header begin
  //
  //header end
  //
  stopMove()
  resetMotion()
  // check robot condition:  ESTOP clear, MANUAL MODE, CALIBRATED=true, ARM POWER=ON
  call initializeRobot()
  userPage()
  cls()
  title(" MOVE TO PARK TOP")
  gotoxy(0,4)
  putln("WAITING:  Press MOVE/HOLD button")
  putln("          to move to Park...")
  // put "HALT" in F8 position
  gotoxy(36,13)
  put("HALT")
  //
  //
  bEnableMonitor=true
  LpPark=jointToPoint(tSensorTool,world,jParkTop)
  movel(LpPark,tSensorTool,mGlobalSpeed)
  //
  // watch for Stay Clear Zone entry, process if required
  // watch for bStopMotion initiated from tskHaltMoveMon()
  bWatchForHalt=true
  do
    // get current position, compare with destination
    LpHere=here(tSensorTool,world)
    LpPark=jointToPoint(tSensorTool,world,jPark)
    LnDistance=abs(distance(LpHere,LpPark))
    delay(0)
  until (LnDistance<=nZoneWatchTol) or (bInsideCube==true) or (bInsideCylinder==true) or (bInsideSphere==true) or (bStopMotion==true)
  //
  if (bInsideCube==false) and (bInsideCylinder==false) and (bInsideSphere==false) and (bStopMotion==false)
    waitEndMove()
    popUpMsg("NOW at PARK TOP...Press OK")
  else
    stopMove()
    resetMotion()
    bStopAllMonitor=true
    popUpMsg("MOTION CANCELLED:  Zone Entered or HALT requested; Monitoring Disabled; Manual Recovery REQUIRED...Press OK")
    //
    // put in motion halt recovery steps here
    //
  endIf
  bEnableMonitor=false
  bWatchForHalt=false
  bStopMotion=false
  //
  //
  //done
  //
end

--- readme.pgx ---
program readme()
begin
  //Title : SLAC RX160L sensor positioning application
  //History:
  //  IOC Release April 2016 by zlentz
  //    change pretty much everything on the remote access side
  //
  //  Changes by klg at some point
  //    reconnect on connection drops, etc.
  //
  //  Release 3 by ???
  //    I don't know what happened here, just filling in the readme gaps
  //
  //  Release 2 <release date here> by Blue Technik LLC
  //    change remote control function from CS8_client to CS8_server
  //      no login function implemented
  //      change sio variable from sioIOChost to sioIOCclient
  //    next addtition
  //    next addition
  //    next addition
  //
  //  Initial Release:
  //    Blue Technik LLC
  //    2507 Watonga Drive, Suite B
  //    Commerce Township, MI  48382
  //    PH:  248-891-8479
  //    FX:  248-366-1560
  //    bt.info@bluetechnik.com
  //    www.bluetechnik.com
  //
  //General description :
  //  This application provides an interactive Teach Pendant Menu method by which SLAC personnel may :
  //  - teach Interaction Point frames (coordinate systems)
  //  - teach Interaction Point sensor Target Points by inputting Azimuth, Elevation, & Radius coordinates
  //    relative to the Interaction Point Frame
  //  - teach "Stay Clear Zones" (cubic, cylindrical, spherical)
  //  - Adjust Target Point orienation in user-selectable resolution
  //  - Teach a Park position
  //  - Teach a Tool Center Point on a tool by two methods
  //
  //
  //Hardware required :
  //  - Robot system    : User robot of choice
  //  - Peripherals     : no peripherals required
  //
  //VAL3 options :
  //  - VAL3 version    : 6.4
  //  - VAL3 licenses   : no licenses required
  //  - VAL3 add-ons    : none
  //
  //Library version     : 6.4.1.0
  //
  //Public variables    : many
  //
  //Included libraries  : monitorAreaEN.............for Definition, Enable/Disable, and monitoring of Stay Clear Zones
  //                      calcToolpEN...............for teaching TCP via reference pointer
  //                      calcTool4pEN..............for teach TCP via 4-point method
  //                      io........................standard Input / Output library
  //
  //Miscellaneous       : ---
  //
  //
  // PROGRAMMING STYLE NOTES
  // Data variable Prefixes
  //  p      = point location
  //  j      = joint location
  //  n      = numerical variable (real and integer)
  //  m      = motion descriptor variable
  //  tr     = trsf transformation value variable
  //  di     = digital input
  //  do     = digital output
  //  b      = boolean variable
  //  f      = robot frame description variable
  //  t      = robot tool transform description variable
  //  sio    = serial I/O port description variable
  //  s    = string variable
  //
  //  LOCAL program variables are identified in their programs
  //  by the prefix "L" before any other variable name values
  //
  //  Subroutine Parameters are identified by the "X" prefix
  //
  //
  //  TCP/IP COMMUNICATIONS TEST METHOD
  //  can test Client-Host communications functionality on user PC with Staubli CS8 Emulator and TeraTerm
  //  /terminal emulator software.
  //    1.  Start CS8 Emulator and run SLAC application to main menu
  //    2.  Start Remote Control.
  //    3.  Start TeraTerm, make New Connection with following settings:
  //        a.  TCP/IP checked ON
  //        b.  Host = whatever is stated at bottom left of CS8 Emulator window, typically = 127.0.0.1
  //        c.  Service = OTHER
  //        d.  TCP Port # = "1301" or whatever the Host port is set to on CS8 Emululator for Host "IOC"
  //        e.  Protocol = UNSPEC
  //    4.  At this point you should see in the TeraTerm window the CS8 response string "LISTENINGX"
  //        /to indicated a good connection has been made.
  //    5.  Change TeraTerm / Setup / Terminal as follows:
  //        a.  New-Line:  Receive = CR+LF
  //        b.  New-Line:  Transmit = CR
  //        c.  Local Echo = ON
  //        d.  All other settings:  leave as defaults
  //    6.  Done with setup.
  //    7.  Enter commands and receive responses to test functionality.
  //
  //
end

--- remCalcHere.pgx ---
program remCalcHere()
  local point pHere
  local trsf trHere
begin
  // Calculate current position in current frame and save to globals
  //
  logMsg("call remCalcHere")
  if nIPNumber==0
    pHere=here(tSensorTool,fIP1)
  else
    pHere=here(tSensorTool,fIP2)
  endIf
  trHere=pHere.trsf
  nXHere=trHere.x
  nYHere=trHere.y
  nZHere=trHere.z
  nRXHere=trHere.rx
  nRYHere=trHere.ry
  nRZHere=trHere.rz
end

--- remCalcHereSph.pgx ---
program remCalcHereSph()
  local num nAzi
  local num nEle
  local num nRad
begin
  // Calculate current position in current frame in
  // spherical coordinates and save to globals
  //
  logMsg("call remCalcHereSph")
  call remCalcHere()

  //calculate azimuthal angle
  if nXHere==0 and nZHere==0
    nAzi=0
  elseIf nXHere==0
    if nZHere>0
      nAzi=0
    else
      nAzi=180
    endIf
  elseIf nZHere==0
    if nXHere>0
      nAzi=90
    else
      nAzi=-90
    endIf
  else
    nAzi=atan(nXHere/nZHere)
    if nZHere<0
      if nXHere>0
        nAzi=nAzi+180
      else
        nAzi=nAzi-180
      endIf
    endIf
  endIf

  //calculate elevation angle
  if nXHere==0 and nYHere==0 and nZHere==0
    nEle=0
  elseIf nXHere==0 and nZHere==0
    if nYHere>0
      nEle=90
    else
      nEle=-90
    endIf
  else
    nEle=atan(nYHere/sqrt(power(nXHere,2)+power(nZHere,2)))
  endIf

  //calculate radius
  nRad=sqrt(power(nXHere,2)+power(nYHere,2)+power(nZHere,2))

  nAzHere=nAzi
  nElHere=nEle
  nRHere=nRad
end

--- remCmdHandler.pgx ---
program remCmdHandler()
  local string LsResponse
  local num nArgs
  local num nArgsReq
  local num nIndex
  local string sArgs
  local string sCmd
  local string sFullCmd
  local string sTemp
begin
  // Command interface with the IOC
  // Parses the command and sends it to the correct subprocess
  //
  sRemMotionCmd=""
  sIOCCommand=""
  nMovArgs=0
  do
    //kill self if remote mode is on and 3 is pressed
    if bRemControlON and isKeyPressed(283)
      bKillRemControl=true
    endIf
    //start tskRemMotion if not running.  Is killed by Client Command String below to
    //stop current motion if any in progress
    if bRemControlON and taskStatus("RemoteMotion")!=1
      putln("RemoteMotion task OFF, starting...")
      logMsg("RemoteMotion task OFF, starting...")
      taskCreate "RemoteMotion",10,remMovHandler()
      wait(taskStatus("RemoteMotion")==1)
      logMsg("RemoteMotion task ON!")
      putln("RemoteMotion task ON!")
    endIf
    // read command string from IOC Host
    sFullCmd=sioIOCclient
    if len(sFullCmd)>0
      // strip off the last CR character of the incoming string
      sFullCmd=delete(sFullCmd,1,len(sFullCmd))
      // separate string into command and arguments. Count the arguments.
      nIndex=find(sFullCmd," ")
      nArgs=0
      if nIndex==-1
        sCmd=sFullCmd
        sArgs=""
      else
        sCmd=left(sFullCmd,nIndex)
        sArgs=delete(sFullCmd,nIndex+1,0)
        sTemp=sArgs
        do
          nArgs=nArgs+1
          nIndex=find(sTemp," ")
          if nIndex!=-1
            sTemp=delete(sTemp,nIndex+1,0)
          endIf
        until nIndex==-1
      endIf
      // even if we're just getting a value, write to the logs
      logMsg("Request "+sFullCmd)
      LsResponse=""
      // print to screen if we're changing sometihng
      sTemp=left(sCmd,3)
      if bRemControlON and (sTemp=="MOV" or sTemp=="SET" or sTemp=="CMD")
        putln(sFullCmd)
      endIf
      if !bRemControlON and sTemp!="GET" and sCmd!="ENABLEREMOTE" and sTemp!="NOT"
        call remErrManual(LsResponse)
      elseIf sTemp=="MOV"
        if bRemMotionBusy==true
          call remErrBusy(LsResponse)
        elseIf isPowered()==false
          call remErrPower(LsResponse)
        else
          sIOCCommand=sArgs
          nMovArgs=nArgs
          sRemMotionCmd=sCmd
        endIf
      else
        switch sCmd
          case "GETPOS"
            call remGetHere(LsResponse)
          break
          case "GETPOSSPH"
            call remGetHereSph(LsResponse)
          break
          case "GETONEPOS"
            nArgsReq=1
            if nArgs==nArgsReq
              call remGetOneHere(sArgs,LsResponse)
            else
              call remErrArgs(sCmd,nArgs,nArgsReq,LsResponse)
            endIf
          break
          case "GETWORLD"
            call remGetWorld(LsResponse)
          break
          case "GETJOINTS"
            call remGetJoints(LsResponse)
          break
          case "CMDDISABLEARM"
            call remDisableArm(LsResponse)
          break
          case "CMDENABLEARM"
            call remEnableArm(LsResponse)
          break
          case "GETARMSTAT"
            call remGetArmStat(LsResponse)
          break
          case "GETESTOP"
            call remGetESTOP(LsResponse)
          break
          case "SETIP"
            nArgsReq=1
            if nArgs==nArgsReq
              call remSetIP(sArgs,LsResponse)
            else
              call remErrArgs(sCmd,nArgs,nArgsReq,LsResponse)
            endIf
          break
          case "GETIP"
            call remGetIP(LsResponse)
          break
          case "SETIPVALS"
            nArgsReq=7
            if nArgs==nArgsReq
              call remSetIPVals(sArgs,LsResponse)
            else
              call remErrArgs(sCmd,nArgs,nArgsReq,LsResponse)
            endIf
          break
          case "GETIPVALS"
            call remGetIPVals(LsResponse)
          break
          case "CMDTRANSIP"
            nArgsReq=3
            if nArgs==nArgsReq
              call remTransIP(sArgs,LsResponse)
            else
              call remErrArgs(sCmd,nArgs,nArgsReq,LsResponse)
            endIf
          break
          case "SETTCPVALS"
            nArgsReq=6
            if nArgs==nArgsReq
              call remSetTCPVals(sArgs,LsResponse)
            else
              call remErrArgs(sCmd,nArgs,nArgsReq,LsResponse)
            endIf
          break
          case "GETTCPVALS"
            call remGetTCPVals(LsResponse)
          break
          case "SETMODE"
            nArgsReq=1
            if nArgs==nArgsReq
              call remSetMode(sArgs,LsResponse)
            else
              call remErrArgs(sCmd,nArgs,nArgsReq,LsResponse)
            endIf
          break
          case "GETMODE"
            call remGetMode(LsResponse)
          break
          case "SETMAXV"
            nArgsReq=1
            if nArgs==nArgsReq
              call remSetMaxV(sArgs,LsResponse)
            else
              call remErrArgs(sCmd,nArgs,nArgsReq,LsResponse)
            endIf
          break
          case "GETMAXV"
            call remGetMaxV(LsResponse)
          break
          case "SETMAXRV"
            nArgsReq=1
            if nArgs==nArgsReq
              call remSetMaxRV(sArgs,LsResponse)
            else
              call remErrArgs(sCmd,nArgs,nArgsReq,LsResponse)
            endIf
          break
          case "GETMAXRV"
            call remGetMaxRV(LsResponse)
          break
          case "SETMAXA"
            nArgsReq=1
            if nArgs==nArgsReq
              call remSetMaxA(sArgs,LsResponse)
            else
              call remErrArgs(sCmd,nArgs,nArgsReq,LsResponse)
            endIf
          break
          case "GETMAXA"
            call remGetMaxA(LsResponse)
          break
          case "SETMAXDIST"
            nArgsReq=1
            if nArgs==nArgsReq
              call remSetMaxDist(sArgs,LsResponse)
            else
              call remErrArgs(sCmd,nArgs,nArgsReq,LsResponse)
            endIf
          break
          case "GETMAXDIST"
            call remGetMaxDist(LsResponse)
          break
          case "GETDMOV"
            call remGetDMOV(LsResponse)
          break
          case "ENABLEREMOTE"
            call remEnableRem(LsResponse)
          break
          case "CMDHALTREMOTE"
            call iocWriteBack("CMDHALTREMOTE")
            bKillRemControl=true
          break
          case "GETREMOTE"
            call remGetRem(LsResponse)
          break
          case "GETERROR"
            call remErrBufferGet(LsResponse)
          break
          case "CMDTEST"
            call remTest(sArgs,LsResponse)
          break

          case "GETPPS"
            call remGetPPS(LsResponse)
          break

          case "NOTPPS"
            nArgsReq=1
            if nArgs==nArgsReq
              call remSetPPS(sArgs,LsResponse)
            else
              call remErrArgs(sCmd,nArgs,nArgsReq,LsResponse)
            endIf
          break

          case "GETHEARTBEAT"
            call remGetHeartbeat(LsResponse)
          break

          case "NOTHEARTBEAT"
            nArgsReq=1
            if nArgs==nArgsReq
              call remSetHeartbeat(sArgs,LsResponse)
            else
              call remErrArgs(sCmd,nArgs,nArgsReq,LsResponse)
            endIf
          break

          case "GETSTAGEPOS"
            call remGetStagePos(LsResponse)
          break

          case "NOTSTAGEPOS"
            nArgsReq=1
            if nArgs==nArgsReq
              call remSetStagePos(sArgs,LsResponse)
            else
              call remErrArgs(sCmd,nArgs,nArgsReq,LsResponse)
            endIf
          break

          case "GETROBOTMODE"
            call remGetRobotMode(LsResponse)
          break



          case "CMDKILLMOTION"
            // cancel the pending command strings & booleans used in other tasks
            sIOCCommand=""
            logMsg("KILLMOTION requested by IOC")
            putln("KILLMOTION requested by IOC")
            bRemMotionBusy=false
            //bEnableMonitor=false
            sRemMotionCmd=""
            //
            // kill Remote Motion task
            putln("STOPPING RemoteMotion task...")
            logMsg("STOPPING RemoteMotion task...")
            taskKill("RemoteMotion")
            wait(taskStatus("RemoteMotion")!=1)
            //
            // stop & reset motion
            stopMove()
            resetMotion()
            putln("RemoteMotion task STOPPED!")
            logMsg("RemoteMotion task STOPPED!")
            putln("MOTION KILLED")
            logMsg("MOTION KILLED")
            LsResponse="CMDKILLMOTION"
          break
          default
            call remErrCmd(sCmd,LsResponse)
          break
        endSwitch
      endIf
      if len(LsResponse)>0
        call iocWriteBack(LsResponse)
      endIf
      //
    endIf
    //this task is killed in tskRemControl()
  until false
  // done
  //
end

--- remDisableArm.pgx ---
program remDisableArm(string& sReturn[] (dimensions=1))
begin
  // Turn the arm power OFF
  //
  logMsg("call remDisableArm")
  stopMove()
  resetMotion()
  disablePower()
  wait(isPowered()==false)
  sReturn="CMDDISABLEARM"
  logMsg("Arm power is DISABLED!")
end

--- remEnableArm.pgx ---
program remEnableArm(string& sReturn[] (dimensions=1))
  local num nTimeout
begin
  // Turn arm power ON
  // Note that this will time out if you were not allowed to do it
  //
  logMsg("call remEnableArm")
  nTimeout=2
  if watch(nPPS>0,nTimeout)
    logMsg("PPS status ready for arm power.")
    if isPowered()==false
      enablePower()
    endIf
    if watch(isPowered(),nTimeout)
      sReturn="CMDENABLEARM"
      logMsg("Arm power ENABLED!")
      putln("Arm power ENABLED!")
    else

      if workingMode()!=4
        call remErrRemoteKey(sReturn)
      else
        call remErrTimeout(nTimeout,sReturn)
      endIf

    endIf


  else
    disablePower()
    call remErrPpTimeout(nTimeout,sReturn)
  endIf


end

--- remEnableRem.pgx ---
program remEnableRem(string& sReturn[] (dimensions=1))
begin
  // Enable remote mode... remotely!
  //
  logMsg("call remEnableRem")
  bRemControlON=true
  sReturn="ENABLEREMOTE"
end

--- remErrArgs.pgx ---
program remErrArgs(string& sCmd[] (dimensions=1), num& nArgs[] (dimensions=1), num nArgsReq (dimensions=1), string& sReturn[] (dimensions=1))
begin
  // Error raised when we recieve the wrong number of arguments.
  //
  logMsg("call remErrArgs")
  sReturn="ERROR 102"
  sReturn=sReturn+": "+sCmd+" received "
  sReturn=sReturn+toString("",nArgs)
  sReturn=sReturn+" args, expected "
  sReturn=sReturn+toString("",nArgsReq)+"."
  putln(sReturn)
  logMsg(sReturn)
end

--- remErrBufferAdd.pgx ---
program remErrBufferAdd(string& sErrMessage[] (dimensions=1))
begin
  //Add an error message to the error buffer
  //Used for errors that may happen long after a command is called
  //e.g. used for end of movement errors because we can't stop the
  //  IOC to wait for them
  //
  logMsg("call remErrBufferAdd")
  sErrBuffer[nErrNext]=sErrMessage
  if nErrNext==nErrBufferSize
    nErrNext=0
  else
    nErrNext=nErrNext+1
  endIf
end

--- remErrBufferGet.pgx ---
program remErrBufferGet(string& sReturn[] (dimensions=1))
begin
  //Get one error from the error buffer, if there is an error
  //
  logMsg("call remErrBufferGet")
  if sErrBuffer[nErrNow]==""
    sReturn="NOERROR"
  else
    sReturn="ERROR "+sErrBuffer[nErrNow]
    putln(sReturn)
    logMsg(sReturn)
    sErrBuffer[nErrNow]=""
    if nErrNow==nErrBufferSize
      nErrNow=0
    else
      nErrNow=nErrNow+1
    endIf
  endIf
end

--- remErrBusy.pgx ---
program remErrBusy(string& sReturn[] (dimensions=1))
begin
  // Error raised when Remote Motion task is busy
  //
  logMsg("call remErrBusy")
  sReturn="ERROR 201"
  sReturn=sReturn+": Move command already active."
  putln(sReturn)
  logMsg(sReturn)
end

--- remErrCmd.pgx ---
program remErrCmd(string& sCmd[] (dimensions=1), string& sReturn[] (dimensions=1))
begin
  // Error raised when the command was invalid
  //
  logMsg("call remErrCmd")
  sReturn="ERROR 101"
  sReturn=sReturn+": Invalid command "+sCmd
  putln(sReturn)
  logMsg(sReturn)
end

--- remErrConfig.pgx ---
program remErrConfig(string& sReturn[] (dimensions=1))
begin
  // Error raised when arm can't reach destination
  //
  logMsg("call remErrConfig")
  sReturn="ERROR 302"
  sReturn=sReturn+": Out of range or bad arm config."
  putln(sReturn)
  logMsg(sReturn)
end

--- remErrFar.pgx ---
program remErrFar(string& sReturn[] (dimensions=1))
begin
  // Error raised when we try to move to a point that is too far
  //
  logMsg("call remErrFar")
  sReturn="ERROR 303: Move distance above limit."
  putln(sReturn)
  logMsg(sReturn)
end

--- remErrInvalid.pgx ---
program remErrInvalid(string sCmd (dimensions=1), string& sArgs[] (dimensions=1), string& sReturn[] (dimensions=1))
begin
  // Error raised when an invalid string argument is recieved
  //
  logMsg("call remErrInvalid")
  sReturn="ERROR 104"
  sReturn=sReturn+": "+sCmd
  sReturn=sReturn+" recieved invalid string arg "
  sReturn=sReturn+sArgs+"."
  putln(sReturn)
  logMsg(sReturn)
end

--- remErrManual.pgx ---
program remErrManual(string& sReturn[] (dimensions=1))
begin
  // Error raised when we attempt a remote-only command in manual mode
  //
  logMsg("call remErrManual")
  sReturn="ERROR 402"
  sReturn=sReturn+": Abort cmd, not in remote mode."
  logMsg(sReturn)
end

--- remErrNum.pgx ---
program remErrNum(string sCmd (dimensions=1), string& sArg[] (dimensions=1), string& sReturn[] (dimensions=1))
begin
  // Error raised when we recieve an non-numerical argument when
  // a number was expected.
  //
  logMsg("call remErrNum")
  sReturn="ERROR 103: "+sCmd+"non-num arg '"+sArg+"'"
  putln(sReturn)
  logMsg(sReturn)
end

--- remErrPower.pgx ---
program remErrPower(string& sReturn[] (dimensions=1))
begin
  // Error raised when we try to move the robot
  // but the arm is not powered
  //
  logMsg("call remErrPower")
  sReturn="ERROR 202"
  sReturn=sReturn+": Arm is not powered."
  putln(sReturn)
  logMsg(sReturn)
end

--- remErrPPTimeout.pgx ---
program remErrPpTimeout(num& nTime[] (dimensions=1), string& sReturn[] (dimensions=1))
begin
  // Error raised when waiting for PPS ready times out
  //
  logMsg("call remErrTimeout")
  sReturn="ERROR 901"
  sReturn=sReturn+": Timeout of PPS ready after "
  sReturn=sReturn+toString("",nTime)+" seconds."
  putln(sReturn)
  logMsg(sReturn)
end

--- remErrRemoteKey.pgx ---
program remErrRemoteKey(string& sReturn[] (dimensions=1))
begin
  // Error raised when a command times out
  //
  logMsg("call remRemoteKey")
  sReturn="ERROR 402"
  sReturn=sReturn+": Select Remote mode using the key box."
  putln(sReturn)
  logMsg(sReturn)
end

--- remErrTimeout.pgx ---
program remErrTimeout(num& nTime[] (dimensions=1), string& sReturn[] (dimensions=1))
begin
  // Error raised when a command times out
  //
  logMsg("call remErrTimeout")
  sReturn="ERROR 401"
  sReturn=sReturn+": Timeout of cmd after "
  sReturn=sReturn+toString("",nTime)+" seconds."
  putln(sReturn)
  logMsg(sReturn)
end

--- remErrZone.pgx ---
program remErrZone(string& sReturn[] (dimensions=1))
  local string sErr
begin
  // Error raised when robot enters a stay clear zone
  // Add to buffer instead of sending to IOC immediately
  //
  logMsg("call remErrZone")
  sErr="301: Entered STAY CLEAR zone!"
  call remErrBufferAdd(sErr)
  putln("ERROR "+sErr)
  logMsg("ERROR "+sErr)
  sReturn=""
end

--- remGetArmStat.pgx ---
program remGetArmStat(string& sReturn[] (dimensions=1))
begin
  // Get whether power is enabled or disabled
  //
  logMsg("call remGetArmStat")
  if isPowered()
    sReturn="GETARMSTAT ENABLED"
  else
    sReturn="GETARMSTAT DISABLED"
  endIf
end

--- remGetDMOV.pgx ---
program remGetDMOV(string& sReturn[] (dimensions=1))
  local string sDmov
begin
  // Return whether or not the robot is done moving.
  //
  logMsg("call remGetDMOV")
  if bRemMotionBusy
    sDmov="FALSE"
  else
    sDmov="TRUE"
  endIf
  sReturn="GETDMOV "+sDmov
end

--- remGetESTOP.pgx ---
program remGetESTOP(string& sReturn[] (dimensions=1))
  local string sEstop
begin
  // Return the ESTOP status
  //
  logMsg("call remGetESTOP")
  switch esStatus()
    case 0
      sEstop="INACTIVE"
    break
    case 1
      sEstop="STOPPED"
    break
    case 2
      sEstop="READY"
    break
  endSwitch
  sReturn="GETESTOP "+sEstop
end

--- remGetHeartbeat.pgx ---
program remGetHeartbeat(string& sReturn[] (dimensions=1))
  local string sCmd
begin
  // Return the PPS status saved in the robot
  //
  logMsg("call remGetHeartBeat")
  sCmd="GETHEARTBEAT"
  call remGetnGlobal(nHeartbeat,sCmd,sReturn)
end

--- remGetHere.pgx ---
program remGetHere(string& sReturn[] (dimensions=1))
begin
  // Return current position in Cartesian coordinates
  //
  logMsg("call remGetHere")
  call remCalcHere()
  sReturn="GETPOS"
  sReturn=sReturn+" "+toString(sNumConv,nXHere)
  sReturn=sReturn+" "+toString(sNumConv,nYHere)
  sReturn=sReturn+" "+toString(sNumConv,nZHere)
  sReturn=sReturn+" "+toString(sNumConv,nRXHere)
  sReturn=sReturn+" "+toString(sNumConv,nRYHere)
  sReturn=sReturn+" "+toString(sNumConv,nRZHere)
end

--- remGetHereSph.pgx ---
program remGetHereSph(string& sReturn[] (dimensions=1))
begin
  // Return current position in spherical coordinates.
  //
  logMsg("call remGetHere")
  call remCalcHereSph()
  sReturn="GETPOSSPH"
  sReturn=sReturn+" "+toString(sNumConv,nAzHere)
  sReturn=sReturn+" "+toString(sNumConv,nElHere)
  sReturn=sReturn+" "+toString(sNumConv,nRHere)
end

--- remGetIP.pgx ---
program remGetIP(string& sReturn[] (dimensions=1))
begin
  // Return which interaction point is active.
  //
  logMsg("call remGetIP")
  sReturn="GETIP "+toString("",nIPNumber)
end

--- remGetIPVals.pgx ---
program remGetIPVals(string& sReturn[] (dimensions=1))
  local trsf trIP
begin
  // Return the values of the active interaction point.
  //
  logMsg("call remGetIPVals")
  if nIPNumber==0
    trIP=fIP1.trsf
  else
    trIP=fIP2.trsf
  endIf
  sReturn="GETIPVALS"
  sReturn=sReturn+" "+toString(sNumConv,trIP.x)
  sReturn=sReturn+" "+toString(sNumConv,trIP.y)
  sReturn=sReturn+" "+toString(sNumConv,trIP.z)
  sReturn=sReturn+" "+toString(sNumConv,trIP.rx)
  sReturn=sReturn+" "+toString(sNumConv,trIP.ry)
  sReturn=sReturn+" "+toString(sNumConv,trIP.rz)
end

--- remGetJoints.pgx ---
program remGetJoints(string& sReturn[] (dimensions=1))
  local joint jPos
begin
  // Return the physical positions of the robot joints
  //
  logMsg("call remGetJoints")
  jPos=herej()
  sReturn="GETJOINTS"
  sReturn=sReturn+" "+toString(sNumConv,jPos.j1)
  sReturn=sReturn+" "+toString(sNumConv,jPos.j2)
  sReturn=sReturn+" "+toString(sNumConv,jPos.j3)
  sReturn=sReturn+" "+toString(sNumConv,jPos.j4)
  sReturn=sReturn+" "+toString(sNumConv,jPos.j5)
  sReturn=sReturn+" "+toString(sNumConv,jPos.j6)
end

--- remGetMaxA.pgx ---
program remGetMaxA(string& sReturn[] (dimensions=1))
  local string sCmd
begin
  // Return maximum allowed acceleration % for remote moves.
  //
  logMsg("call remGetMaxA")
  sCmd="GETMAXA"
  call remGetnGlobal(nMaxAccel,sCmd,sReturn)
end

--- remGetMaxDist.pgx ---
program remGetMaxDist(string& sReturn[] (dimensions=1))
  local string sCmd
begin
  // Return max dist in a single move step for remote moves (mm)
  //
  logMsg("call remGetMaxDist")
  sCmd="GETMAXDIST"
  call remGetnGlobal(nMaxAccel,sCmd,sReturn)
end

--- remGetMaxRV.pgx ---
program remGetMaxRV(string& sReturn[] (dimensions=1))
  local string sCmd
begin
  // Return maximum allowed rotational velocity in deg/s for remote moves.
  //
  logMsg("call remGetMaxRV")
  sCmd="GETMAXRV"
  call remGetnGlobal(nMaxAccel,sCmd,sReturn)
end

--- remGetMaxV.pgx ---
program remGetMaxV(string& sReturn[] (dimensions=1))
  local string sCmd
begin
  // Return max translational velocity for remote moves (mm/s)
  //
  logMsg("call remGetMaxV")
  sCmd="GETMAXV"
  call remGetnGlobal(nMaxAccel,sCmd,sReturn)
end

--- remGetMode.pgx ---
program remGetMode(string& sReturn[] (dimensions=1))
  local string sMode
begin
  // Return the movement mode for remote moves
  //
  logMsg("call remGetMode")
  if bMoveLinear
    sMode="LINEAR"
  else
    sMode="OPTIMAL"
  endIf
  sReturn="GETMODE "+sMode
end

--- remGetnGlobal.pgx ---
program remGetnGlobal(num& nGlobal[] (dimensions=1), string& sCmd[] (dimensions=1), string& sReturn[] (dimensions=1))
begin
  // Get an arbitrary global value and return it
  //
  logMsg("call remGetnGlobal")
  sReturn=sCmd+" "+toString(sNumConv,nGlobal)
end

--- remGetOneHere.pgx ---
program remGetOneHere(string& sArgs[] (dimensions=1), string& sReturn[] (dimensions=1))
  local joint jHere
  local num nPos
begin
  // Return just one position.
  //
  logMsg("call remGetOneHere")
  call remCalcHereSph()
  jHere=herej()
  sReturn="GETONEPOS "+sArgs+" "
  switch sArgs
    case "X"
      nPos=nXHere
    break
    case "Y"
      nPos=nYHere
    break
    case "Z"
      nPos=nZHere
    break
    case "RX"
      nPos=nRXHere
    break
    case "RY"
      nPos=nRYHere
    break
    case "RZ"
      nPos=nRZHere
    break
    case "AZI"
      nPos=nAzHere
    break
    case "ELE"
      nPos=nElHere
    break
    case "RAD"
      nPos=nRHere
    break
    case "J1"
      nPos=jHere.j1
    break
    case "J2"
      nPos=jHere.j2
    break
    case "J3"
      nPos=jHere.j3
    break
    case "J4"
      nPos=jHere.j4
    break
    case "J5"
      nPos=jHere.j5
    break
    case "J6"
      nPos=jHere.j6
    break
    default
      call remErrInvalid("GETONEPOS",sArgs,sReturn)
    break
  endSwitch
  sReturn=sReturn+toString(sNumConv,nPos)
end

--- remGetPPS.pgx ---
program remGetPPS(string& sReturn[] (dimensions=1))
  local string sCmd
begin
  // Return the PPS status saved in the robot
  //
  logMsg("call remGetPPS")
  sCmd="GETPPS"
  call remGetnGlobal(nPPS,sCmd,sReturn)
end

--- remGetRem.pgx ---
program remGetRem(string& sReturn[] (dimensions=1))
begin
  // Return current remote control state
  //
  logMsg("call remGetRem")
  if bRemControlON
    sReturn="REMOTE"
  else
    sReturn="MANUAL"
  endIf
  sReturn="GETREMOTE "+sReturn
end

--- remGetRobotMode.pgx ---
program remGetRobotMode(string& sReturn[] (dimensions=1))
  local string sCmd
begin
  // Return the PPS status saved in the robot
  //
  logMsg("call remGetRobotMode")
  sCmd="GETROBOTMODE"
  call remGetnGlobal(nRobotMode,sCmd,sReturn)
end

--- remGetStagePos.pgx ---
program remGetStagePos(string& sReturn[] (dimensions=1))
  local string sCmd
begin
  // Return the PPS status saved in the robot
  //
  logMsg("call remGetStagePos")
  sCmd="GETSTAGEPOS"
  call remGetnGlobal(nStagePos,sCmd,sReturn)
end

--- remGetTCPVals.pgx ---
program remGetTCPVals(string& sReturn[] (dimensions=1))
  local trsf trTCP
begin
  // Return the Cartesian values of the TCP
  //
  logMsg("call remSetIPVals")
  trTCP=tSensorTool.trsf
  sReturn="GETTCPVALS"
  sReturn=sReturn+" "+toString(sNumConv,trTCP.x)
  sReturn=sReturn+" "+toString(sNumConv,trTCP.y)
  sReturn=sReturn+" "+toString(sNumConv,trTCP.z)
  sReturn=sReturn+" "+toString(sNumConv,trTCP.rx)
  sReturn=sReturn+" "+toString(sNumConv,trTCP.ry)
  sReturn=sReturn+" "+toString(sNumConv,trTCP.rz)
end

--- remGetWorld.pgx ---
program remGetWorld(string& sReturn[] (dimensions=1))
  local point pHere
  local trsf trHere
begin
  // Return the world position values, ignoring the current frame.
  //
  logMsg("call remGetWorld")
  pHere=here(tSensorTool,world)
  trHere=pHere.trsf
  sReturn="GETWORLD"
  sReturn=sReturn+" "+toString(sNumConv,trHere.x)
  sReturn=sReturn+" "+toString(sNumConv,trHere.y)
  sReturn=sReturn+" "+toString(sNumConv,trHere.z)
  sReturn=sReturn+" "+toString(sNumConv,trHere.rx)
  sReturn=sReturn+" "+toString(sNumConv,trHere.ry)
  sReturn=sReturn+" "+toString(sNumConv,trHere.rz)
end

--- remMovAxis.pgx ---
program remMovAxis(string& sArgs[] (dimensions=1), string& sReturn[] (dimensions=1))
  local bool bOk
  local num nIndex
  local num nVal
  local string sAxis
  local string sVal
  local trsf trDest
begin
  // Move robot to a specific point along one axis,
  // keeping positions along other axes in the Cartesian
  // coordinate system static.
  //
  // Arguments are "AXIS NUMBER" e.g. "X 35"
  //
  logMsg("call remMovAxis")
  //parse args, expecting axis label and a number.
  //We already know we have exactly 2 args.
  nIndex=find(sArgs," ")
  sAxis=left(sArgs,nIndex)
  sVal=delete(sArgs,nIndex+1,0)
  toNum(sVal,nVal,bOk)
  if bOk
    call remCalcHere()
    trDest={nXHere,nYHere,nZHere,nRXHere,nRYHere,nRZHere}
    switch sAxis
      case "X"
        trDest.x=nVal
      break
      case "Y"
        trDest.y=nVal
      break
      case "Z"
        trDest.z=nVal
      break
      case "RX"
        trDest.rx=nVal
      break
      case "RY"
        trDest.ry=nVal
      break
      case "RZ"
        trDest.rz=nVal
      break
      default
        call remErrInvalid("MOVAXIS",sAxis,sReturn)
        return
      break
    endSwitch
    call remMovPoint(trDest,sReturn)
  else
    call remErrNum("MOVAXIS",sVal,sReturn)
  endIf
end

--- remMovAZELRA.pgx ---
program remMovAZELRA(string& sArgs[] (dimensions=1), string& sReturn[] (dimensions=1))
  local bool bOk
  local num nAzi
  local num nEle
  local num nLoop
  local num nRad
  local num nVal
  local string sArgsLoop
begin
  // Move to a specified point in spherical coordinates
  //
  // Arguments are "AZ EL RA"
  //
  logMsg("call remMovAZELRA")
  //break down our 3 args and make sure they are numbers
  nLoop=0
  sArgsLoop=sArgs
  while nLoop<3
    sArgsLoop=toNum(sArgsLoop,nVal,bOk)
    if bOk
      switch nLoop
        case 0
          nAzi=nVal
        break
        case 1
          nEle=nVal
        break
        case 2
          nRad=nVal
        break
      endSwitch
      nLoop=nLoop+1
    else
      call remErrNum("MOVAZELRA",sArgs,sReturn)
      return
    endIf
  endWhile
  call remMovSph(nAzi,nEle,nRad,sReturn)
end

--- remMovBase.pgx ---
program remMovBase(point& pDest[] (dimensions=1), string& sReturn[] (dimensions=1))
  local bool bMovOk
  local joint jDest
  local joint jHere
  local mdesc mUserSpeed
  local num nDistance
  local string sGoal
  local trsf trGoal
begin
  // Move to a given point, handling movement
  // parameters and stay clear zones.
  //
  logMsg("call remMovBase")
  //first, check if movement is possible.
  jHere=herej()
  bMovOk=pointToJoint(tSensorTool,jHere,pDest,jDest)
  if bMovOk
    //check if we're moving too far (user set max dist)
    nDistance=abs(distance(here(tSensorTool,world),pDest))
    //put a line to say where we're going to
    trGoal=pDest.trsf
    sGoal="Moving "+toString(sNumConv,nDistance)+" mm to ("
    sGoal=sGoal+toString(sNumConv,trGoal.x)+", "
    sGoal=sGoal+toString(sNumConv,trGoal.y)+", "
    sGoal=sGoal+toString(sNumConv,trGoal.z)+", "
    sGoal=sGoal+toString(sNumConv,trGoal.rx)+", "
    sGoal=sGoal+toString(sNumConv,trGoal.ry)+", "
    sGoal=sGoal+toString(sNumConv,trGoal.rz)+")"
    putln(sGoal)
    logMsg(sGoal)
    if nDistance<nMaxDist
      mUserSpeed={nMaxAccel,100,nMaxAccel,nMaxVelo,nMaxRVelo,off,50,50}
      call iocWriteBack("ARMMOVING")
      putln("ARM MOVING")
      logMsg("ARM MOVING")
      bEnableMonitor=true
      if bMoveLinear
        movel(pDest,tSensorTool,mUserSpeed)
      else
        movej(jDest,tSensorTool,mUserSpeed)
      endIf
      //watch for stay clear zones
      do
        nDistance=abs(distance(here(tSensorTool,world),pDest))
        delay(0)
        //stop checking if done or if zone is violated
      until nDistance<=nZoneWatchTol or bInsideCube or bInsideCylinder or bInsideSphere
      //stop and raise error if we violated a stay clear zone
      if bInsideCube or bInsideCylinder or bInsideSphere
        stopMove()
        resetMotion()
        bStopAllMonitor=true
        call remErrZone(sReturn)
      else
        waitEndMove()
        sReturn=""
      endIf
      putln("ARM DONE MOVING")
      logMsg("ARM DONE MOVING")
      bEnableMonitor=false
    else
      //destination was too far, so we raise an error
      call remErrFar(sReturn)
    endIf
  else
    //destination was impossible, so we raise an error
    call remErrConfig(sReturn)
  endIf
end

--- remMovHandler.pgx ---
program remMovHandler()
  local bool LbError
  local string LsCommandString
  local string LsCubeValsIOC
  local string LsCylValsIOC
  local string LsESTOPIOC
  local string LsError
  local string LsIOCCommand
  local string LsJointValsIOC
  local string LsLength
  local string LsResponse
  local string LsSphValsIOC
  local string LsTCPValsIOC
begin
  // Handle movement commands
  //
  while true
    if sRemMotionCmd!=""
      bRemMotionBusy=true
      switch sRemMotionCmd
        case "MOVXYZ"
          if nMovArgs==6
            call remMovXYZ(sIOCCommand,LsResponse)
          else
            call remErrArgs(sRemMotionCmd,nMovArgs,6,LsResponse)
          endIf
        break
        case "MOVAZELRA"
          if nMovArgs==3
            call remMovAZELRA(sIOCCommand,LsResponse)
          else
            call remErrArgs(sRemMotionCmd,nMovArgs,3,LsResponse)
          endIf
        break
        case "MOVAXIS"
          if nMovArgs==2
            call remMovAxis(sIOCCommand,LsResponse)
          else
            call remErrArgs(sRemMotionCmd,nMovArgs,2,LsResponse)
          endIf
        break
        case "MOVSPHAXIS"
          if nMovArgs==2
            call remMovSphAxis(sIOCCommand,LsResponse)
          else
            call remErrArgs(sRemMotionCmd,nMovArgs,2,LsResponse)
          endIf
        break
        case "MOVJOINT"
          if nMovArgs==6
            call remMovJoint(sIOCCommand,LsResponse)
          else
            call remErrArgs(sRemMotionCmd,nMovArgs,6,LsResponse)
          endIf
        break
        case "MOVJOINTAXIS"
          if nMovArgs==2
            call remMovJointAxis(sIOCCommand,LsResponse)
          else
            call remErrArgs(sRemMotionCmd,nMovArgs,2,LsResponse)
          endIf
        break
        default
          call remErrCmd(sRemMotionCmd,LsResponse)
        break
      endSwitch
      if len(LsResponse)>0
        call iocWriteBack(LsResponse)
      endIf
      sRemMotionCmd=""
      sIOCCommand=""
      nMovArgs=0
      bRemMotionBusy=false
    endIf
    delay(0)
  endWhile
end

--- remMovJoint.pgx ---
program remMovJoint(string& sArgs[] (dimensions=1), string& sReturn[] (dimensions=1))
  local bool bOk
  local joint jDest
  local num nLoop
  local num nVal
  local point pDest
  local string sArgsLoop
begin
  // Move to the designated point.
  //
  // Arguments are "J1 J2 J3 J4 J5 J6"
  //
  logMsg("call remMovJoint")
  //break down our 6 args and make sure they are numbers
  jDest={0,0,0,0,0,0}
  nLoop=0
  sArgsLoop=sArgs
  while nLoop<6
    sArgsLoop=toNum(sArgsLoop,nVal,bOk)
    if bOk
      switch nLoop
        case 0
          jDest.j1=nVal
        break
        case 1
          jDest.j2=nVal
        break
        case 2
          jDest.j3=nVal
        break
        case 3
          jDest.j4=nVal
        break
        case 4
          jDest.j5=nVal
        break
        case 5
          jDest.j6=nVal
        break
      endSwitch
      nLoop=nLoop+1
    else
      call remErrNum("MOVJOINT",sArgs,sReturn)
      return
    endIf
  endWhile
  if nIPNumber==0
    pDest=jointToPoint(tSensorTool,fIP1,jDest)
  else
    pDest=jointToPoint(tSensorTool,fIP2,jDest)
  endIf
  call remMovBase(pDest,sReturn)
end

--- remMovJointAxis.pgx ---
program remMovJointAxis(string& sArgs[] (dimensions=1), string& sReturn[] (dimensions=1))
  local bool bOk
  local joint jDest
  local num nIndex
  local num nVal
  local point pDest
  local string sAxis
  local string sVal
begin
  //Move just one joint
  //Arguments are "j pos" where j is J1, J2, J3, J4, J5, or J6 and pos is the goal
  //
  logMsg("call remMovJointAxis")
  nIndex=find(sArgs," ")
  sAxis=left(sArgs,nIndex)
  sVal=delete(sArgs,nIndex+1,0)
  toNum(sVal,nVal,bOk)
  if bOk
    jDest=herej()
    switch sAxis
      case "J1"
        jDest.j1=nVal
      break
      case "J2"
        jDest.j2=nVal
      break
      case "J3"
        jDest.j3=nVal
      break
      case "J4"
        jDest.j4=nVal
      break
      case "J5"
        jDest.j5=nVal
      break
      case "J6"
        jDest.j6=nVal
      break
      default
        call remErrInvalid("MOVJOINTAXIS",sAxis,sReturn)
        return
      break
    endSwitch
    if nIPNumber==0
      pDest=jointToPoint(tSensorTool,fIP1,jDest)
    else
      pDest=jointToPoint(tSensorTool,fIP2,jDest)
    endIf
    call remMovBase(pDest,sReturn)
  else
    call remErrNum("MOVJOINTAXIS",sVal,sReturn)
  endIf
end

--- remMovPoint.pgx ---
program remMovPoint(trsf& trXYZ[] (dimensions=1), string& sReturn[] (dimensions=1))
  local point pDest
begin
  // Given coordinates, construct the point object for
  // remMoveBase in current frame of reference
  //
  logMsg("call remMovPoint")
  if nIPNumber==0
    pDest=compose(pIP1NullPoint,fIP1,trXYZ)
  else
    pDest=compose(pIP2NullPoint,fIP2,trXYZ)
  endIf
  call remMovBase(pDest,sReturn)
end

--- remMovSph.pgx ---
public program remMovSph(num& nAzi[], num& nEle[], num& nRad[], string& sReturn[])
  local trsf trXYZ
begin
  // Move to designated point in spherical coordinates
  // Point detector to the center of rotation
  //
  logMsg("call remMovSph")
  // Transpose trsf to get correct x, y, z and rotational values
  //trXYZ={0,0,0,0,0,0}
  //trXYZ=trXYZ*{0,0,0,0,nAzi,0}
  //trXYZ=trXYZ*{0,0,0,-nEle,0,0}
  //trXYZ=trXYZ*{0,0,nRad,0,0,0}
  //trXYZ=trXYZ*{0,0,0,-180,0,0}

      // new definitions to match SLAC spec math
    trXYZ={0,0,0,0,0,0}
    // Add AZ component:  rotate about fIPn_+Yaxis
   trXYZ=trXYZ*{0,0,0,0,nAzi,0}
    // Add EL component:  rotate about fIPn_+Z'axis
   trXYZ=trXYZ*{0,0,0,-nEle,0,0}
    // Add RA component:  translate along fIPn+X'axis
    trXYZ=trXYZ*{0,0,nRad,0,0,0}
    // now transform the point so that +Zaxis points back to fIPn
   trXYZ=trXYZ*{0,0,0,0,-180,0}
   //trXYZ.config={sfree,efree,wfree}


  call remMovPoint(trXYZ,sReturn)
end

--- remMovSphAxis.pgx ---
program remMovSphAxis(string& sArgs[] (dimensions=1), string& sReturn[] (dimensions=1))
  local bool bOk
  local num nAzi
  local num nEle
  local num nIndex
  local num nRad
  local num nVal
  local string sAxis
  local string sVal
begin
  // Move to a designated point along an axis in
  // spherical coordinates, keeping other axes constant.
  //
  // arguments are "AXIS POS", e.g. "RAD 1000"
  //
  logMsg("call remMovSphAxis")
  //parse args, expecting axis label and a number.
  //We already know we have exactly 2 args.
  nIndex=find(sArgs," ")
  sAxis=left(sArgs,nIndex)
  sVal=delete(sArgs,nIndex+1,0)
  toNum(sVal,nVal,bOk)
  if bOk
    call remCalcHereSph()
    nAzi=nAzHere
    nEle=nElHere
    nRad=nRHere
    switch sAxis
      case "AZI"
        nAzi=nVal
      break
      case "ELE"
        nEle=nVal
      break
      case "RAD"
        nRad=nVal
      break
      default
        call remErrInvalid("MOVSPHAXIS",sAxis,sReturn)
        return
      break
    endSwitch
    call remMovSph(nAzi,nEle,nRad,sReturn)
  else
    call remErrNum("MOVSPHAXIS",sVal,sReturn)
  endIf
end

--- remMovXYZ.pgx ---
program remMovXYZ(string& sArgs[] (dimensions=1), string& sReturn[] (dimensions=1))
  local bool bOk
  local num nLoop
  local num nVal
  local string sArgsLoop
  local trsf trDest
begin
  // Move to the designated point.
  //
  // Arguments are "X Y Z RX RY RZ"
  //
  logMsg("call remMovXYZ")
  //break down our 6 args and make sure they are numbers
  trDest={0,0,0,0,0,0}
  nLoop=0
  sArgsLoop=sArgs
  while nLoop<6
    sArgsLoop=toNum(sArgsLoop,nVal,bOk)
    if bOk
      switch nLoop
        case 0
          trDest.x=nVal
        break
        case 1
          trDest.y=nVal
        break
        case 2
          trDest.z=nVal
        break
        case 3
          trDest.rx=nVal
        break
        case 4
          trDest.ry=nVal
        break
        case 5
          trDest.rz=nVal
        break
      endSwitch
      nLoop=nLoop+1
    else
      call remErrNum("MOVXYZ",sArgs,sReturn)
      return
    endIf
  endWhile
  call remMovPoint(trDest,sReturn)
end

--- remSetHeartbeat.pgx ---
program remSetHeartbeat(string& sArgs[] (dimensions=1), string& sReturn[] (dimensions=1))
begin
  // Set the PPS status in the robot
  //
  logMsg("call remSetHeatbeat")
  call remSetnGlobal(sArgs,nHeartbeat,0,5000,"NOTHEARTBEAT",sReturn)
end

--- remSetIP.pgx ---
program remSetIP(string& sArgs[] (dimensions=1), string& sReturn[] (dimensions=1))
  local bool bOk
  local num nIP
begin
  // Pick the active IP, 0 or 1.
  //
  logMsg("call remSetIP with args "+sArgs)
  toNum(left(sArgs,1),nIP,bOk)
  if bOk
    if nIP==0
      nIPNumber=0
    else
      nIPNumber=1
    endIf
    sReturn="SETIP "+toString("",nIPNumber)
  else
    call remErrNum("SETIP",sArgs,sReturn)
  endIf
end

--- remSetIPVals.pgx ---
program remSetIPVals(string& sArgs[] (dimensions=1), string& sReturn[] (dimensions=1))
  local bool bOk
  local num nArg
  local num nIP
  local num nTemp
  local trsf trIP
begin
  // Change the values of the active interaction point.
  //
  // Arguments are "X Y Z RX RY RZ"
  //
  logMsg("call remSetIPVals")
  nArg=0
  trIP={0,0,0,0,0,0}
  while nArg<7
    sArgs=toNum(sArgs,nTemp,bOk)
    if bOk
      switch nArg
        case 0
          nIP=nTemp
        break
        case 1
          trIP.x=nTemp
        break
        case 2
          trIP.y=nTemp
        break
        case 3
          trIP.z=nTemp
        break
        case 4
          trIP.rx=nTemp
        break
        case 5
          trIP.ry=nTemp
        break
        case 6
          trIP.rz=nTemp
        break
      endSwitch
      nArg=nArg+1
    else
      call remErrNum("SETIPVALS",sArgs,sReturn)
      return
    endIf
  endWhile
  if nIP==0
    fIP1.trsf=trIP
  else
    fIP2.trsf=trIP
  endIf
  sReturn="SETIPVALS"
end

--- remSetMaxA.pgx ---
program remSetMaxA(string& sArgs[] (dimensions=1), string& sReturn[] (dimensions=1))
  local num bOk
  local num nVal
begin
  // Set the maximum allowed Acceleration in %
  //
  logMsg("call remSetMaxA")
  call remSetnGlobal(sArgs,nMaxAccel,0,100,"SETMAXA",sReturn)
end

--- remSetMaxDist.pgx ---
program remSetMaxDist(string& sArgs[] (dimensions=1), string& sReturn[] (dimensions=1))
begin
  // Set the maximum allowed move dist in mm
  //
  logMsg("call remSetMaxDist")
  call remSetnGlobal(sArgs,nMaxDist,0,5000,"SETMAXDIST",sReturn)
end

--- remSetMaxRV.pgx ---
program remSetMaxRV(string& sArgs[] (dimensions=1), string& sReturn[] (dimensions=1))
  local bool bOk
  local num nVal
begin
  // Set the maximum allowed rotational velocity in deg/s
  //
  logMsg("call remSetMaxRV")
  call remSetnGlobal(sArgs,nMaxRVelo,0,45,"SETMAXRV",sReturn)
end

--- remSetMaxV.pgx ---
program remSetMaxV(string& sArgs[] (dimensions=1), string& sReturn[] (dimensions=1))
  local num bOk
  local num nVal
begin
  // Set the maximum allowed translational velocity in mm/s.
  //
  logMsg("call remSetMaxV")
  call remSetnGlobal(sArgs,nMaxVelo,0,200,"SETMAXV",sReturn)
end

--- remSetMode.pgx ---
program remSetMode(string& sArgs[] (dimensions=1), string& sReturn[] (dimensions=1))
begin
  // Set the remote movement mode to LINEAR or OPTIMAL
  //
  logMsg("call remSetMode")
  if sArgs=="LINEAR"
    bMoveLinear=true
  elseIf sArgs=="OPTIMAL"
    bMoveLinear=false
  else
    call remErrInvalid("SETMODE",sArgs,sReturn)
    return
  endIf
  sReturn="SETMODE "+sArgs
end

--- remSetnGlobal.pgx ---
program remSetnGlobal(string& sArgs[] (dimensions=1), num& nGlobal[] (dimensions=1), num nMin (dimensions=1), num nMax (dimensions=1), string sCmd (dimensions=1), string& sReturn[] (dimensions=1))
  local bool bOk
  local num nVal
begin
  // Read a command to set an arbitrary global value,
  // and respond accordingly.
  //
  logMsg("call remSetnGlobal")
  toNum(sArgs,nVal,bOk)
  if bOk
    if nVal<nMin
      nVal=nMin
    elseIf nVal>nMax
      nVal=nMax
    endIf
    nGlobal=nVal
    sReturn=sCmd+" "+toString(sNumConv,nGlobal)
  else
    call remErrNum(sCmd,sArgs,sReturn)
  endIf
end

